// Mitsubishi GX Works2 project: GCP-712CRB_1910022_210518R   PLC: Q03UDV
// SECS

PROGRAM 01INITI
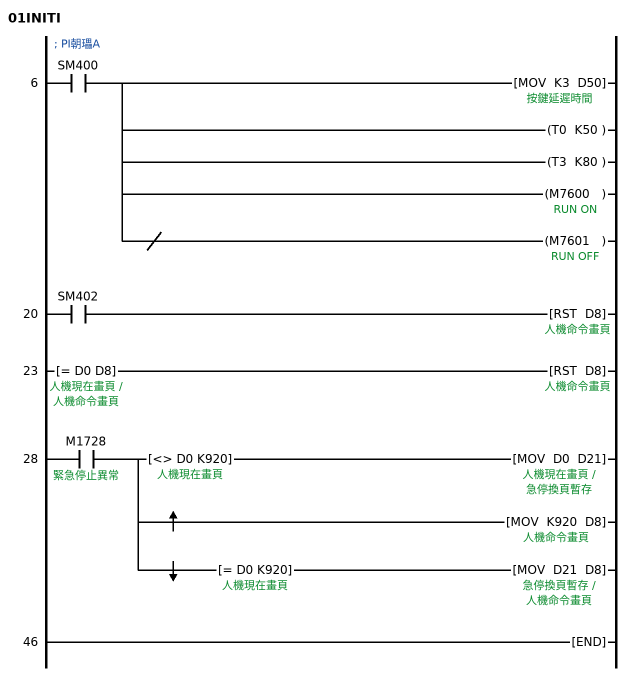
; PI朝瓃Α
6     LD      SM400
      MOV     K3 D50  ; 按鍵延遲時間
      OUT     T0 K50
      OUT     T3 K80
      OUT     M7600  ; RUN ON
      INV
      OUT     M7601  ; RUN OFF
20    LD      SM402
      RST     D8  ; 人機命令畫頁
23    LD=     D0 D8  ; 人機現在畫頁 / 人機命令畫頁
      RST     D8  ; 人機命令畫頁
28    LD      M1728  ; 緊急停止異常
      MPS
      AND<>   D0 K920  ; 人機現在畫頁
      MOV     D0 D21  ; 急停換頁暫存
      MRD
      MEP
      MOV     K920 D8
      MPP
      MEF
      AND=    D0 K920  ; 人機現在畫頁
      MOV     D21 D8
46    END
END_PROGRAM

PROGRAM 02FUNC
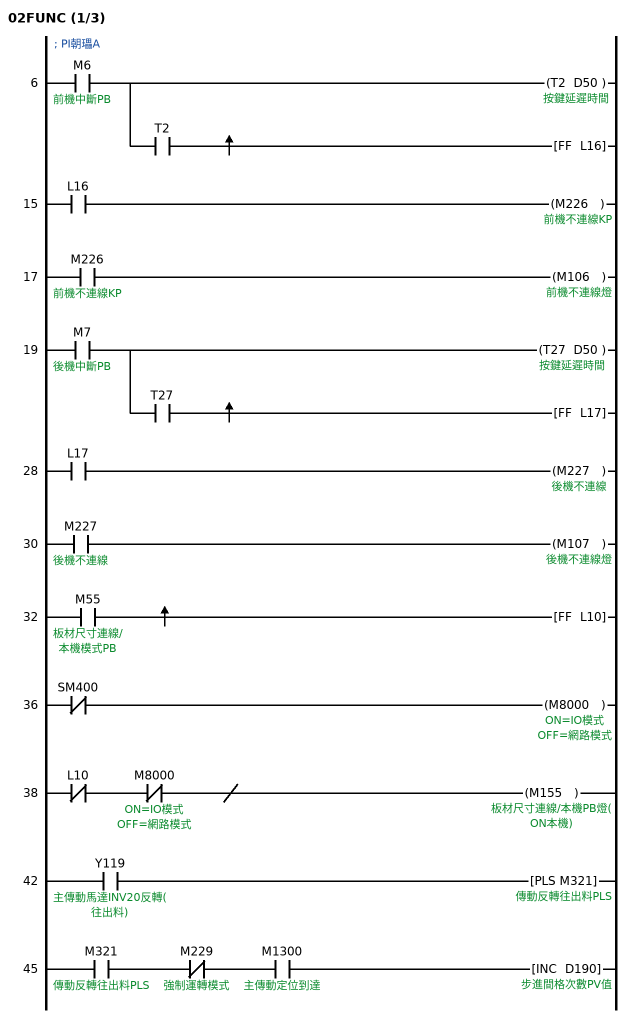
; PI朝瓃Α
6     LD      M6  ; 前機中斷PB
      OUT     T2 D50  ; 按鍵延遲時間
      AND     T2
      MEP
      FF      L16
15    LD      L16
      OUT     M226  ; 前機不連線KP
17    LD      M226  ; 前機不連線KP
      OUT     M106  ; 前機不連線燈
19    LD      M7  ; 後機中斷PB
      OUT     T27 D50  ; 按鍵延遲時間
      AND     T27
      MEP
      FF      L17
28    LD      L17
      OUT     M227  ; 後機不連線
30    LD      M227  ; 後機不連線
      OUT     M107  ; 後機不連線燈
32    LD      M55  ; 板材尺寸連線/本機模式PB
      MEP
      FF      L10
36    LDI     SM400
      OUT     M8000  ; ON=IO模式 OFF=網路模式
38    LDI     L10
      ANI     M8000  ; ON=IO模式 OFF=網路模式
      INV
      OUT     M155  ; 板材尺寸連線/本機PB燈(ON本機)
42    LD      Y119  ; 主傳動馬達INV20反轉(往出料)
      PLS     M321  ; 傳動反轉往出料PLS
45    LD      M321  ; 傳動反轉往出料PLS
      ANI     M229  ; 強制運轉模式
      AND     M1300  ; 主傳動定位到達
      INC     D190  ; 步進間格次數PV值
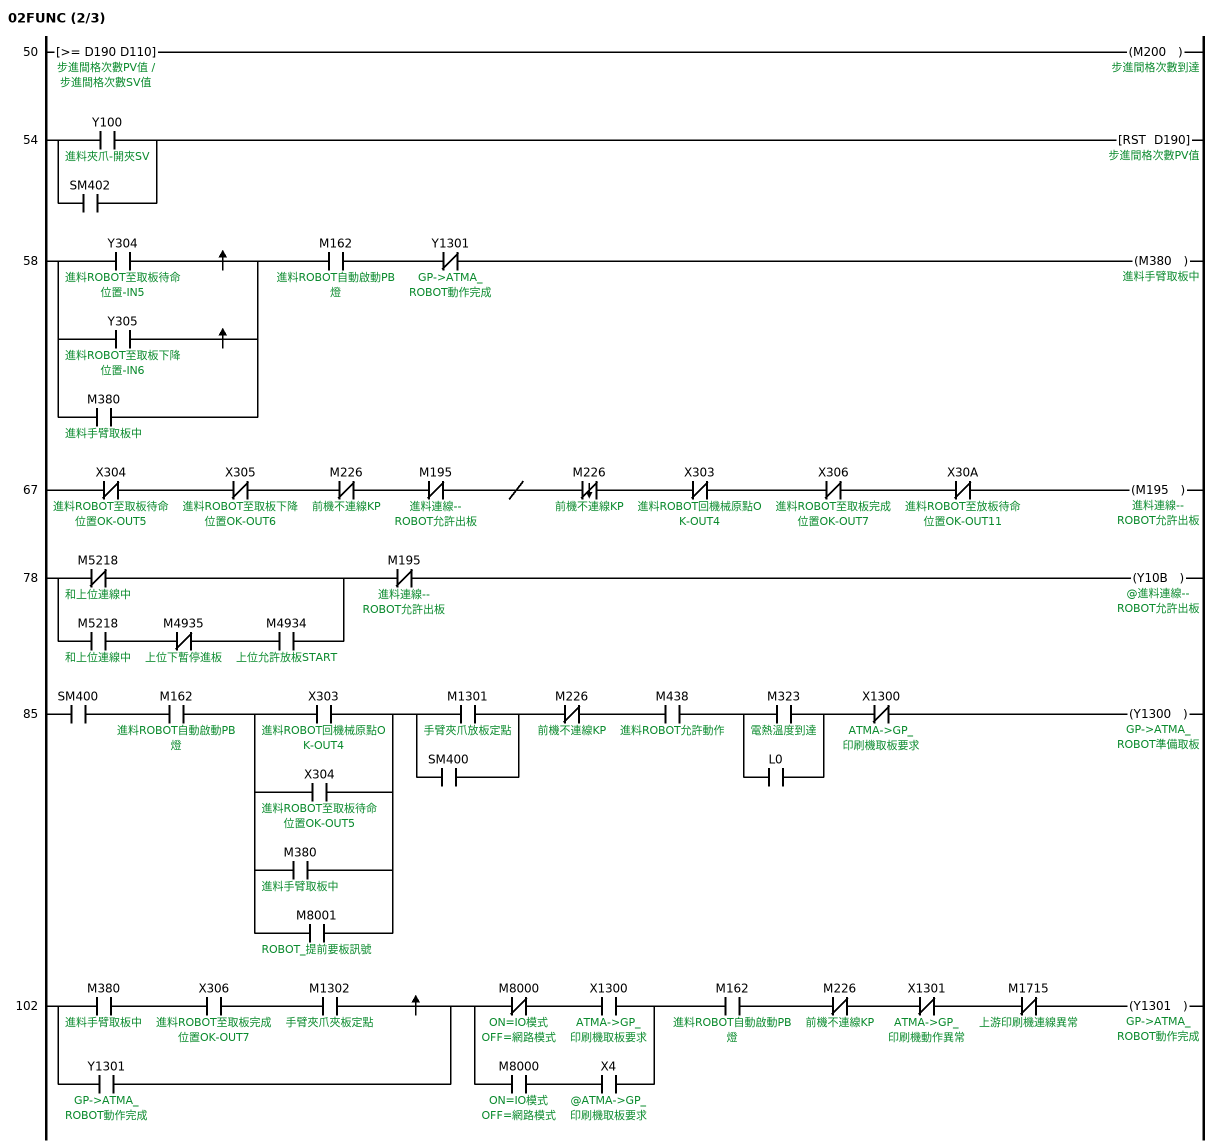
50    LD>=    D190 D110  ; 步進間格次數PV值 / 步進間格次數SV值
      OUT     M200  ; 步進間格次數到達
54    LD      Y100  ; 進料夾爪-開夾SV
      OR      SM402
      RST     D190  ; 步進間格次數PV值
58    LD      Y304  ; 進料ROBOT至取板待命位置-IN5
      MEP
      LD      Y305  ; 進料ROBOT至取板下降位置-IN6
      MEP
      ORB
      OR      M380  ; 進料手臂取板中
      AND     M162  ; 進料ROBOT自動啟動PB燈
      ANI     Y1301  ; GP->ATMA_ROBOT動作完成
      OUT     M380  ; 進料手臂取板中
67    LDI     X304  ; 進料ROBOT至取板待命位置OK-OUT5
      ANI     X305  ; 進料ROBOT至取板下降位置OK-OUT6
      ANI     M226  ; 前機不連線KP
      ANI     M195  ; 進料連線--ROBOT允許出板
      INV
      ANDFI   M226  ; 前機不連線KP
      ANI     X303  ; 進料ROBOT回機械原點OK-OUT4
      ANI     X306  ; 進料ROBOT至取板完成位置OK-OUT7
      ANI     X30A  ; 進料ROBOT至放板待命位置OK-OUT11
      OUT     M195  ; 進料連線--ROBOT允許出板
78    LDI     M5218  ; 和上位連線中
      LD      M5218  ; 和上位連線中
      ANI     M4935  ; 上位下暫停進板
      AND     M4934  ; 上位允許放板START
      ORB
      ANI     M195  ; 進料連線--ROBOT允許出板
      OUT     Y10B  ; @進料連線--ROBOT允許出板
85    LD      SM400
      AND     M162  ; 進料ROBOT自動啟動PB燈
      LD      X303  ; 進料ROBOT回機械原點OK-OUT4
      OR      X304  ; 進料ROBOT至取板待命位置OK-OUT5
      OR      M380  ; 進料手臂取板中
      OR      M8001  ; ROBOT_提前要板訊號
      ANB
      LD      M1301  ; 手臂夾爪放板定點
      OR      SM400
      ANB
      ANI     M226  ; 前機不連線KP
      AND     M438  ; 進料ROBOT允許動作
      LD      M323  ; 電熱溫度到達
      OR      L0
      ANB
      ANI     X1300  ; ATMA->GP_印刷機取板要求
      OUT     Y1300  ; GP->ATMA_ROBOT準備取板
102   LD      M380  ; 進料手臂取板中
      AND     X306  ; 進料ROBOT至取板完成位置OK-OUT7
      AND     M1302  ; 手臂夾爪夾板定點
      MEP
      OR      Y1301  ; GP->ATMA_ROBOT動作完成
      LDI     M8000  ; ON=IO模式 OFF=網路模式
      AND     X1300  ; ATMA->GP_印刷機取板要求
      LD      M8000  ; ON=IO模式 OFF=網路模式
      AND     X4  ; @ATMA->GP_印刷機取板要求
      ORB
      ANB
      AND     M162  ; 進料ROBOT自動啟動PB燈
      ANI     M226  ; 前機不連線KP
      ANI     X1301  ; ATMA->GP_印刷機動作異常
      ANI     M1715  ; 上游印刷機連線異常
      OUT     Y1301  ; GP->ATMA_ROBOT動作完成
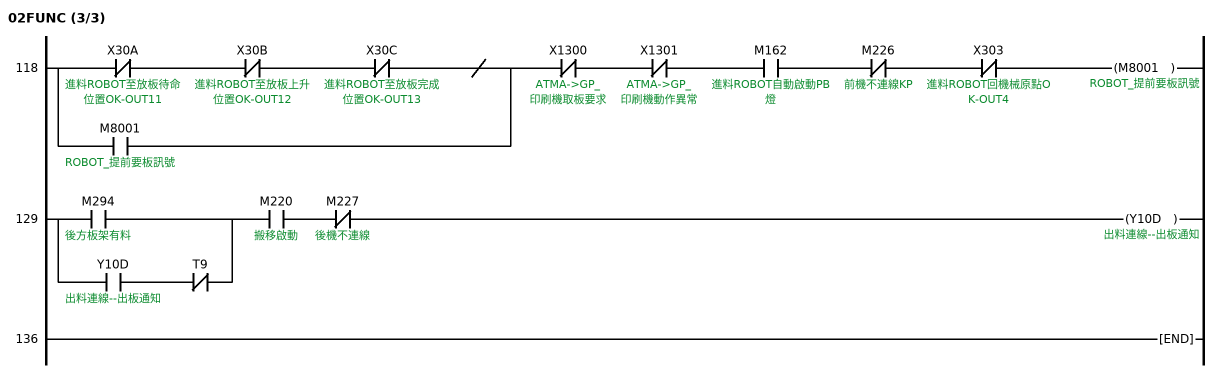
118   LDI     X30A  ; 進料ROBOT至放板待命位置OK-OUT11
      ANI     X30B  ; 進料ROBOT至放板上升位置OK-OUT12
      ANI     X30C  ; 進料ROBOT至放板完成位置OK-OUT13
      INV
      OR      M8001  ; ROBOT_提前要板訊號
      ANI     X1300  ; ATMA->GP_印刷機取板要求
      ANI     X1301  ; ATMA->GP_印刷機動作異常
      AND     M162  ; 進料ROBOT自動啟動PB燈
      ANI     M226  ; 前機不連線KP
      ANI     X303  ; 進料ROBOT回機械原點OK-OUT4
      OUT     M8001  ; ROBOT_提前要板訊號
129   LD      M294  ; 後方板架有料
      LD      Y10D  ; 出料連線--出板通知
      ANI     T9
      ORB
      AND     M220  ; 搬移啟動
      ANI     M227  ; 後機不連線
      OUT     Y10D  ; 出料連線--出板通知
136   END
END_PROGRAM

PROGRAM 03ORIGIN
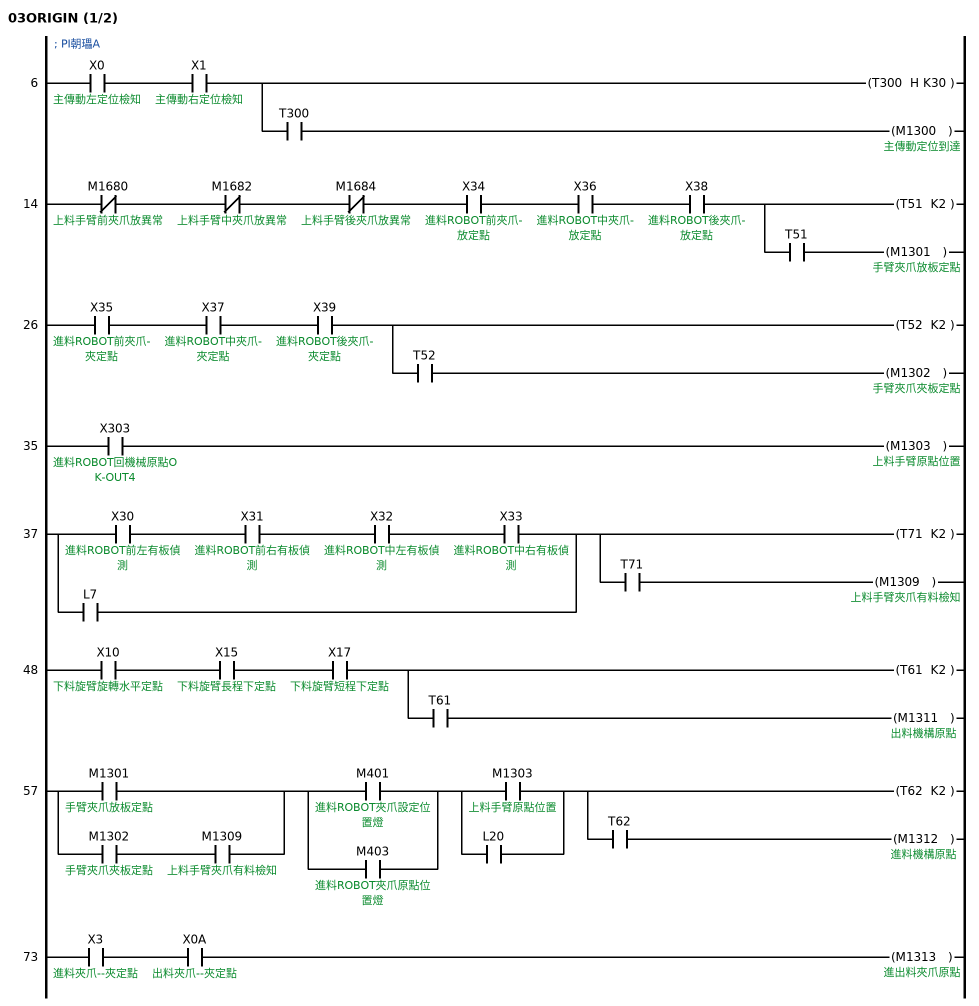
; PI朝瓃Α
6     LD      X0  ; 主傳動左定位檢知
      AND     X1  ; 主傳動右定位檢知
      OUTH    T300 K30
      AND     T300
      OUT     M1300  ; 主傳動定位到達
14    LDI     M1680  ; 上料手臂前夾爪放異常
      ANI     M1682  ; 上料手臂中夾爪放異常
      ANI     M1684  ; 上料手臂後夾爪放異常
      AND     X34  ; 進料ROBOT前夾爪-放定點
      AND     X36  ; 進料ROBOT中夾爪-放定點
      AND     X38  ; 進料ROBOT後夾爪-放定點
      OUT     T51 K2
      AND     T51
      OUT     M1301  ; 手臂夾爪放板定點
26    LD      X35  ; 進料ROBOT前夾爪-夾定點
      AND     X37  ; 進料ROBOT中夾爪-夾定點
      AND     X39  ; 進料ROBOT後夾爪-夾定點
      OUT     T52 K2
      AND     T52
      OUT     M1302  ; 手臂夾爪夾板定點
35    LD      X303  ; 進料ROBOT回機械原點OK-OUT4
      OUT     M1303  ; 上料手臂原點位置
37    LD      X30  ; 進料ROBOT前左有板偵測
      AND     X31  ; 進料ROBOT前右有板偵測
      AND     X32  ; 進料ROBOT中左有板偵測
      AND     X33  ; 進料ROBOT中右有板偵測
      OR      L7
      OUT     T71 K2
      AND     T71
      OUT     M1309  ; 上料手臂夾爪有料檢知
48    LD      X10  ; 下料旋臂旋轉水平定點
      AND     X15  ; 下料旋臂長程下定點
      AND     X17  ; 下料旋臂短程下定點
      OUT     T61 K2
      AND     T61
      OUT     M1311  ; 出料機構原點
57    LD      M1301  ; 手臂夾爪放板定點
      LD      M1302  ; 手臂夾爪夾板定點
      AND     M1309  ; 上料手臂夾爪有料檢知
      ORB
      LD      M401  ; 進料ROBOT夾爪設定位置燈
      OR      M403  ; 進料ROBOT夾爪原點位置燈
      ANB
      LD      M1303  ; 上料手臂原點位置
      OR      L20
      ANB
      OUT     T62 K2
      AND     T62
      OUT     M1312  ; 進料機構原點
73    LD      X3  ; 進料夾爪--夾定點
      AND     X0A  ; 出料夾爪--夾定點
      OUT     M1313  ; 進出料夾爪原點
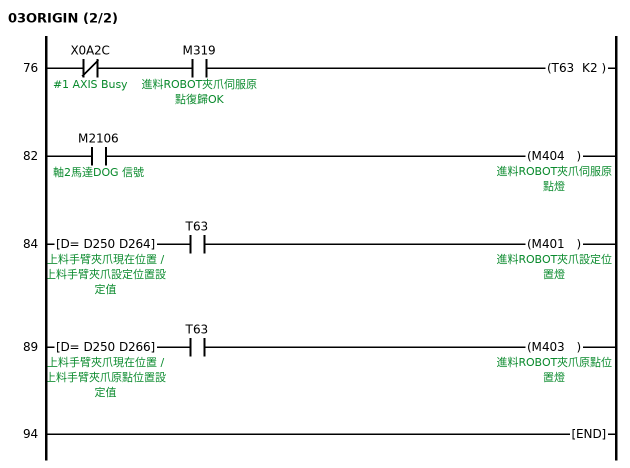
76    LDI     X0A2C  ; #1 AXIS Busy
      AND     M319  ; 進料ROBOT夾爪伺服原點復歸OK
      OUT     T63 K2
82    LD      M2106  ; 軸2馬達DOG 信號
      OUT     M404  ; 進料ROBOT夾爪伺服原點燈
84    LDD=    D250 D264  ; 上料手臂夾爪現在位置 / 上料手臂夾爪設定位置設定值
      AND     T63
      OUT     M401  ; 進料ROBOT夾爪設定位置燈
89    LDD=    D250 D266  ; 上料手臂夾爪現在位置 / 上料手臂夾爪原點位置設定值
      AND     T63
      OUT     M403  ; 進料ROBOT夾爪原點位置燈
94    END
END_PROGRAM

PROGRAM 04LOAD
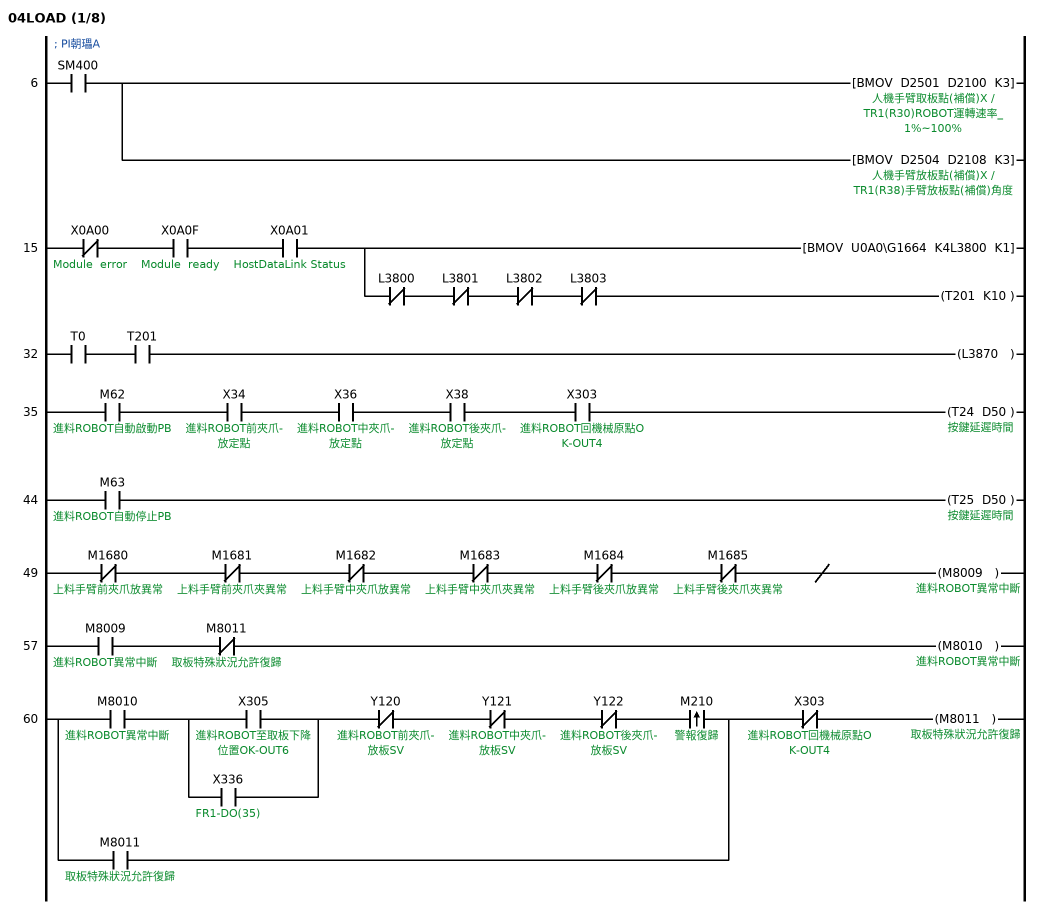
; PI朝瓃Α
6     LD      SM400
      BMOV    D2501 D2100 K3  ; 人機手臂取板點(補償)X / TR1(R30)ROBOT運轉速率_1%~100%
      BMOV    D2504 D2108 K3  ; 人機手臂放板點(補償)X / TR1(R38)手臂放板點(補償)角度
15    LDI     X0A00  ; Module  error
      AND     X0A0F  ; Module  ready
      AND     X0A01  ; HostDataLink Status
      BMOV    U0A0\G1664 K4L3800 K1
      ANI     L3800
      ANI     L3801
      ANI     L3802
      ANI     L3803
      OUT     T201 K10
32    LD      T0
      AND     T201
      OUT     L3870
35    LD      M62  ; 進料ROBOT自動啟動PB
      AND     X34  ; 進料ROBOT前夾爪-放定點
      AND     X36  ; 進料ROBOT中夾爪-放定點
      AND     X38  ; 進料ROBOT後夾爪-放定點
      AND     X303  ; 進料ROBOT回機械原點OK-OUT4
      OUT     T24 D50  ; 按鍵延遲時間
44    LD      M63  ; 進料ROBOT自動停止PB
      OUT     T25 D50  ; 按鍵延遲時間
49    LDI     M1680  ; 上料手臂前夾爪放異常
      ANI     M1681  ; 上料手臂前夾爪夾異常
      ANI     M1682  ; 上料手臂中夾爪放異常
      ANI     M1683  ; 上料手臂中夾爪夾異常
      ANI     M1684  ; 上料手臂後夾爪放異常
      ANI     M1685  ; 上料手臂後夾爪夾異常
      INV
      OUT     M8009  ; 進料ROBOT異常中斷
57    LD      M8009  ; 進料ROBOT異常中斷
      ANI     M8011  ; 取板特殊狀況允許復歸
      OUT     M8010  ; 進料ROBOT異常中斷
60    LD      M8010  ; 進料ROBOT異常中斷
      LD      X305  ; 進料ROBOT至取板下降位置OK-OUT6
      OR      X336  ; FR1-DO(35)
      ANB
      ANI     Y120  ; 進料ROBOT前夾爪-放板SV
      ANI     Y121  ; 進料ROBOT中夾爪-放板SV
      ANI     Y122  ; 進料ROBOT後夾爪-放板SV
      ANDP    M210  ; 警報復歸
      OR      M8011  ; 取板特殊狀況允許復歸
      ANI     X303  ; 進料ROBOT回機械原點OK-OUT4
      OUT     M8011  ; 取板特殊狀況允許復歸
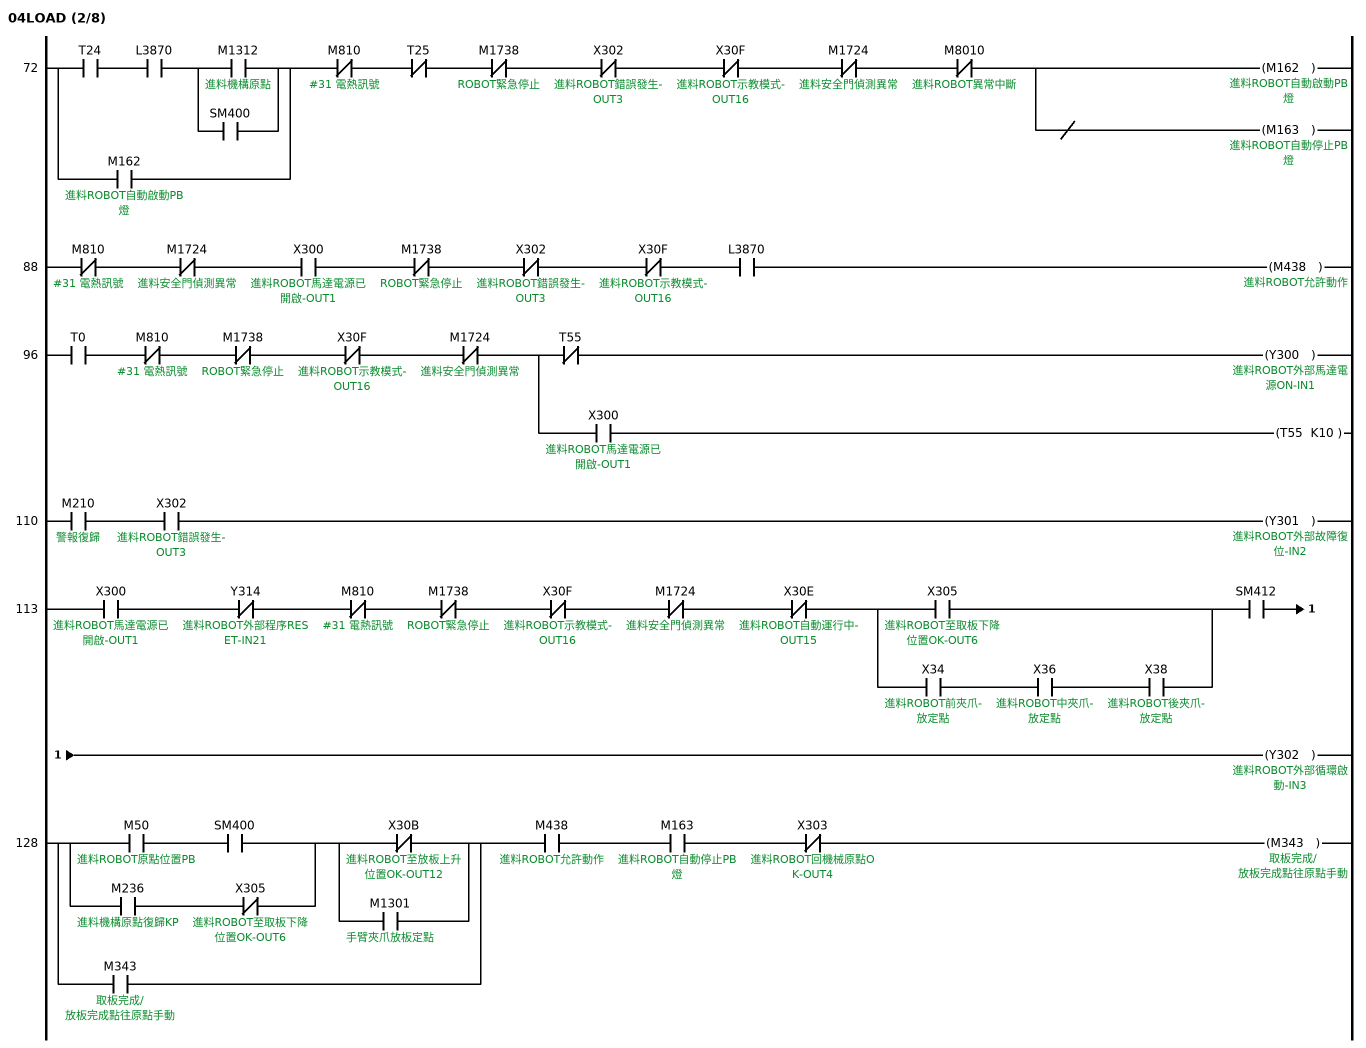
72    LD      T24
      AND     L3870
      LD      M1312  ; 進料機構原點
      OR      SM400
      ANB
      OR      M162  ; 進料ROBOT自動啟動PB燈
      ANI     M810  ; #31 電熱訊號
      ANI     T25
      ANI     M1738  ; ROBOT緊急停止
      ANI     X302  ; 進料ROBOT錯誤發生-OUT3
      ANI     X30F  ; 進料ROBOT示教模式-OUT16
      ANI     M1724  ; 進料安全門偵測異常
      ANI     M8010  ; 進料ROBOT異常中斷
      OUT     M162  ; 進料ROBOT自動啟動PB燈
      INV
      OUT     M163  ; 進料ROBOT自動停止PB燈
88    LDI     M810  ; #31 電熱訊號
      ANI     M1724  ; 進料安全門偵測異常
      AND     X300  ; 進料ROBOT馬達電源已開啟-OUT1
      ANI     M1738  ; ROBOT緊急停止
      ANI     X302  ; 進料ROBOT錯誤發生-OUT3
      ANI     X30F  ; 進料ROBOT示教模式-OUT16
      AND     L3870
      OUT     M438  ; 進料ROBOT允許動作
96    LD      T0
      ANI     M810  ; #31 電熱訊號
      ANI     M1738  ; ROBOT緊急停止
      ANI     X30F  ; 進料ROBOT示教模式-OUT16
      ANI     M1724  ; 進料安全門偵測異常
      MPS
      ANI     T55
      OUT     Y300  ; 進料ROBOT外部馬達電源ON-IN1
      MPP
      AND     X300  ; 進料ROBOT馬達電源已開啟-OUT1
      OUT     T55 K10
110   LD      M210  ; 警報復歸
      AND     X302  ; 進料ROBOT錯誤發生-OUT3
      OUT     Y301  ; 進料ROBOT外部故障復位-IN2
113   LD      X300  ; 進料ROBOT馬達電源已開啟-OUT1
      ANI     Y314  ; 進料ROBOT外部程序RESET-IN21
      ANI     M810  ; #31 電熱訊號
      ANI     M1738  ; ROBOT緊急停止
      ANI     X30F  ; 進料ROBOT示教模式-OUT16
      ANI     M1724  ; 進料安全門偵測異常
      ANI     X30E  ; 進料ROBOT自動運行中-OUT15
      LD      X305  ; 進料ROBOT至取板下降位置OK-OUT6
      LD      X34  ; 進料ROBOT前夾爪-放定點
      AND     X36  ; 進料ROBOT中夾爪-放定點
      AND     X38  ; 進料ROBOT後夾爪-放定點
      ORB
      ANB
      AND     SM412
      OUT     Y302  ; 進料ROBOT外部循環啟動-IN3
128   LD      M50  ; 進料ROBOT原點位置PB
      AND     SM400
      LD      M236  ; 進料機構原點復歸KP
      ANI     X305  ; 進料ROBOT至取板下降位置OK-OUT6
      ORB
      LDI     X30B  ; 進料ROBOT至放板上升位置OK-OUT12
      OR      M1301  ; 手臂夾爪放板定點
      ANB
      OR      M343  ; 取板完成/放板完成點往原點手動
      AND     M438  ; 進料ROBOT允許動作
      AND     M163  ; 進料ROBOT自動停止PB燈
      ANI     X303  ; 進料ROBOT回機械原點OK-OUT4
      OUT     M343  ; 取板完成/放板完成點往原點手動
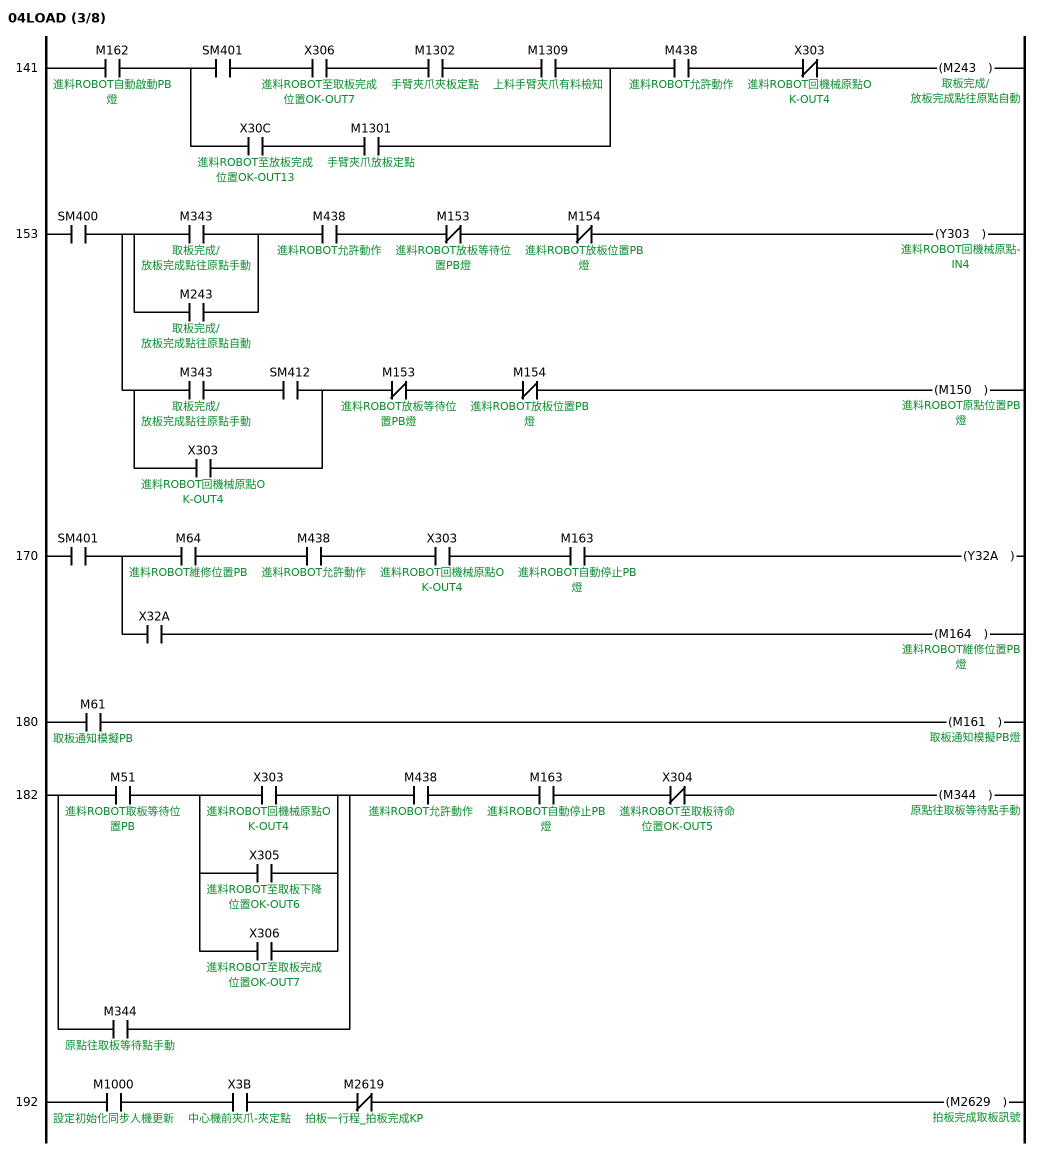
141   LD      M162  ; 進料ROBOT自動啟動PB燈
      LD      SM401
      AND     X306  ; 進料ROBOT至取板完成位置OK-OUT7
      AND     M1302  ; 手臂夾爪夾板定點
      AND     M1309  ; 上料手臂夾爪有料檢知
      LD      X30C  ; 進料ROBOT至放板完成位置OK-OUT13
      AND     M1301  ; 手臂夾爪放板定點
      ORB
      ANB
      AND     M438  ; 進料ROBOT允許動作
      ANI     X303  ; 進料ROBOT回機械原點OK-OUT4
      OUT     M243  ; 取板完成/放板完成點往原點自動
153   LD      SM400
      MPS
      LD      M343  ; 取板完成/放板完成點往原點手動
      OR      M243  ; 取板完成/放板完成點往原點自動
      ANB
      AND     M438  ; 進料ROBOT允許動作
      ANI     M153  ; 進料ROBOT放板等待位置PB燈
      ANI     M154  ; 進料ROBOT放板位置PB燈
      OUT     Y303  ; 進料ROBOT回機械原點-IN4
      MPP
      LD      M343  ; 取板完成/放板完成點往原點手動
      AND     SM412
      OR      X303  ; 進料ROBOT回機械原點OK-OUT4
      ANB
      ANI     M153  ; 進料ROBOT放板等待位置PB燈
      ANI     M154  ; 進料ROBOT放板位置PB燈
      OUT     M150  ; 進料ROBOT原點位置PB燈
170   LD      SM401
      MPS
      AND     M64  ; 進料ROBOT維修位置PB
      AND     M438  ; 進料ROBOT允許動作
      AND     X303  ; 進料ROBOT回機械原點OK-OUT4
      AND     M163  ; 進料ROBOT自動停止PB燈
      OUT     Y32A
      MPP
      AND     X32A
      OUT     M164  ; 進料ROBOT維修位置PB燈
180   LD      M61  ; 取板通知模擬PB
      OUT     M161  ; 取板通知模擬PB燈
182   LD      M51  ; 進料ROBOT取板等待位置PB
      LD      X303  ; 進料ROBOT回機械原點OK-OUT4
      OR      X305  ; 進料ROBOT至取板下降位置OK-OUT6
      OR      X306  ; 進料ROBOT至取板完成位置OK-OUT7
      ANB
      OR      M344  ; 原點往取板等待點手動
      AND     M438  ; 進料ROBOT允許動作
      AND     M163  ; 進料ROBOT自動停止PB燈
      ANI     X304  ; 進料ROBOT至取板待命位置OK-OUT5
      OUT     M344  ; 原點往取板等待點手動
192   LD      M1000  ; 設定初始化同步人機更新
      AND     X3B  ; 中心機前夾爪-夾定點
      ANI     M2619  ; 拍板一行程_拍板完成KP
      OUT     M2629  ; 拍板完成取板訊號
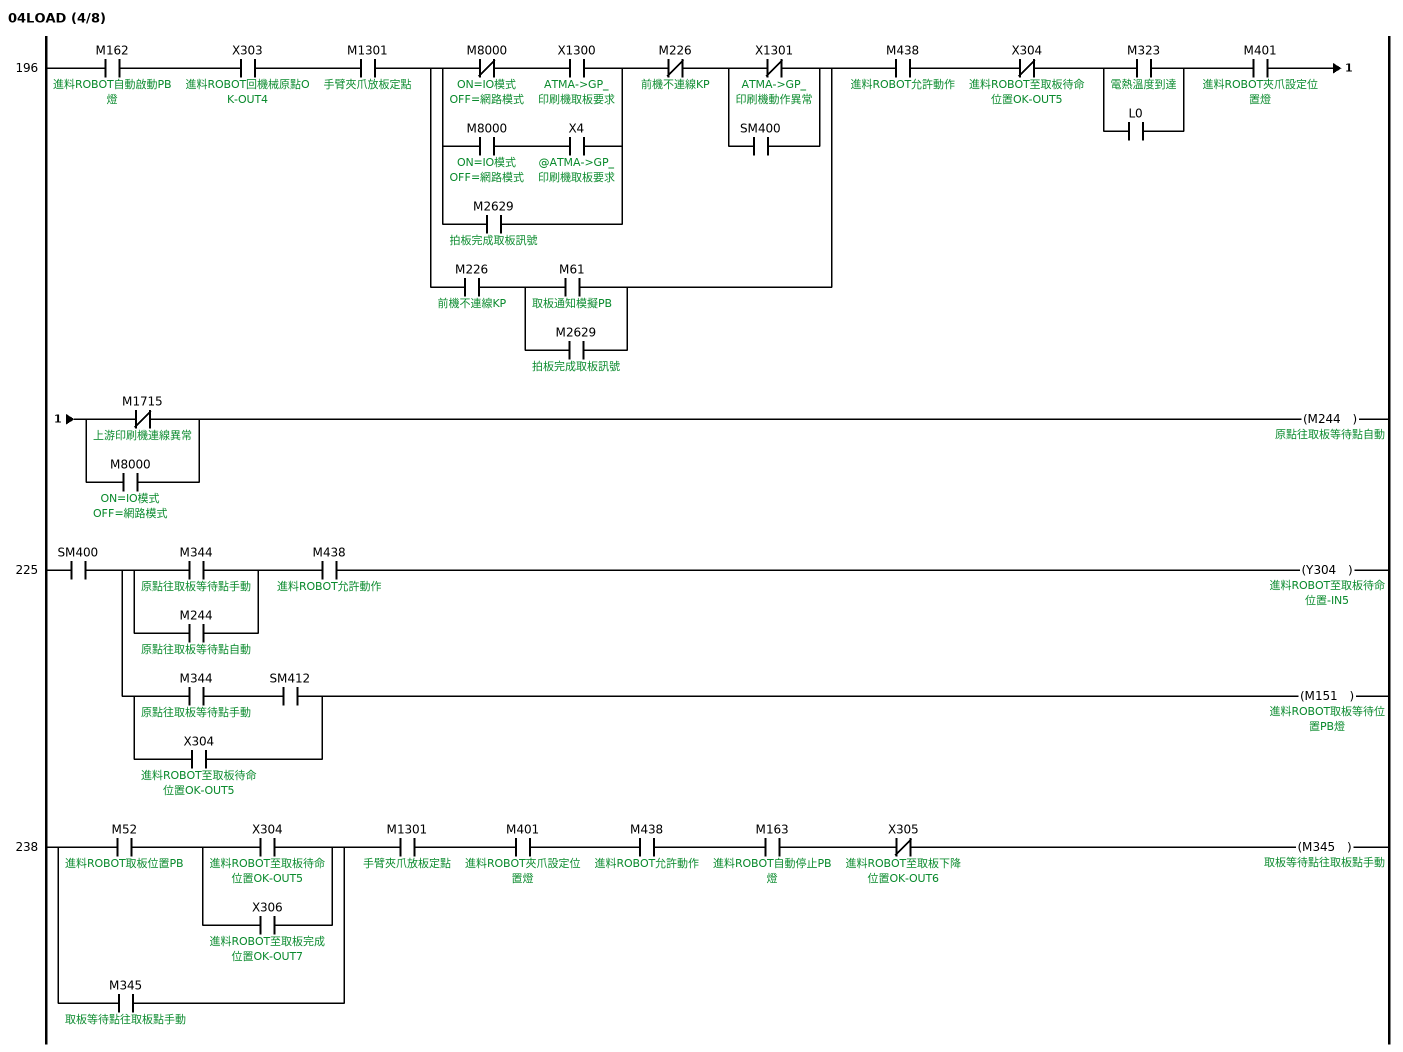
196   LD      M162  ; 進料ROBOT自動啟動PB燈
      AND     X303  ; 進料ROBOT回機械原點OK-OUT4
      AND     M1301  ; 手臂夾爪放板定點
      LDI     M8000  ; ON=IO模式 OFF=網路模式
      AND     X1300  ; ATMA->GP_印刷機取板要求
      LD      M8000  ; ON=IO模式 OFF=網路模式
      AND     X4  ; @ATMA->GP_印刷機取板要求
      ORB
      OR      M2629  ; 拍板完成取板訊號
      ANI     M226  ; 前機不連線KP
      LDI     X1301  ; ATMA->GP_印刷機動作異常
      OR      SM400
      ANB
      LD      M226  ; 前機不連線KP
      LD      M61  ; 取板通知模擬PB
      OR      M2629  ; 拍板完成取板訊號
      ANB
      ORB
      ANB
      AND     M438  ; 進料ROBOT允許動作
      ANI     X304  ; 進料ROBOT至取板待命位置OK-OUT5
      LD      M323  ; 電熱溫度到達
      OR      L0
      ANB
      AND     M401  ; 進料ROBOT夾爪設定位置燈
      LDI     M1715  ; 上游印刷機連線異常
      OR      M8000  ; ON=IO模式 OFF=網路模式
      ANB
      OUT     M244  ; 原點往取板等待點自動
225   LD      SM400
      MPS
      LD      M344  ; 原點往取板等待點手動
      OR      M244  ; 原點往取板等待點自動
      ANB
      AND     M438  ; 進料ROBOT允許動作
      OUT     Y304  ; 進料ROBOT至取板待命位置-IN5
      MPP
      LD      M344  ; 原點往取板等待點手動
      AND     SM412
      OR      X304  ; 進料ROBOT至取板待命位置OK-OUT5
      ANB
      OUT     M151  ; 進料ROBOT取板等待位置PB燈
238   LD      M52  ; 進料ROBOT取板位置PB
      LD      X304  ; 進料ROBOT至取板待命位置OK-OUT5
      OR      X306  ; 進料ROBOT至取板完成位置OK-OUT7
      ANB
      OR      M345  ; 取板等待點往取板點手動
      AND     M1301  ; 手臂夾爪放板定點
      AND     M401  ; 進料ROBOT夾爪設定位置燈
      AND     M438  ; 進料ROBOT允許動作
      AND     M163  ; 進料ROBOT自動停止PB燈
      ANI     X305  ; 進料ROBOT至取板下降位置OK-OUT6
      OUT     M345  ; 取板等待點往取板點手動
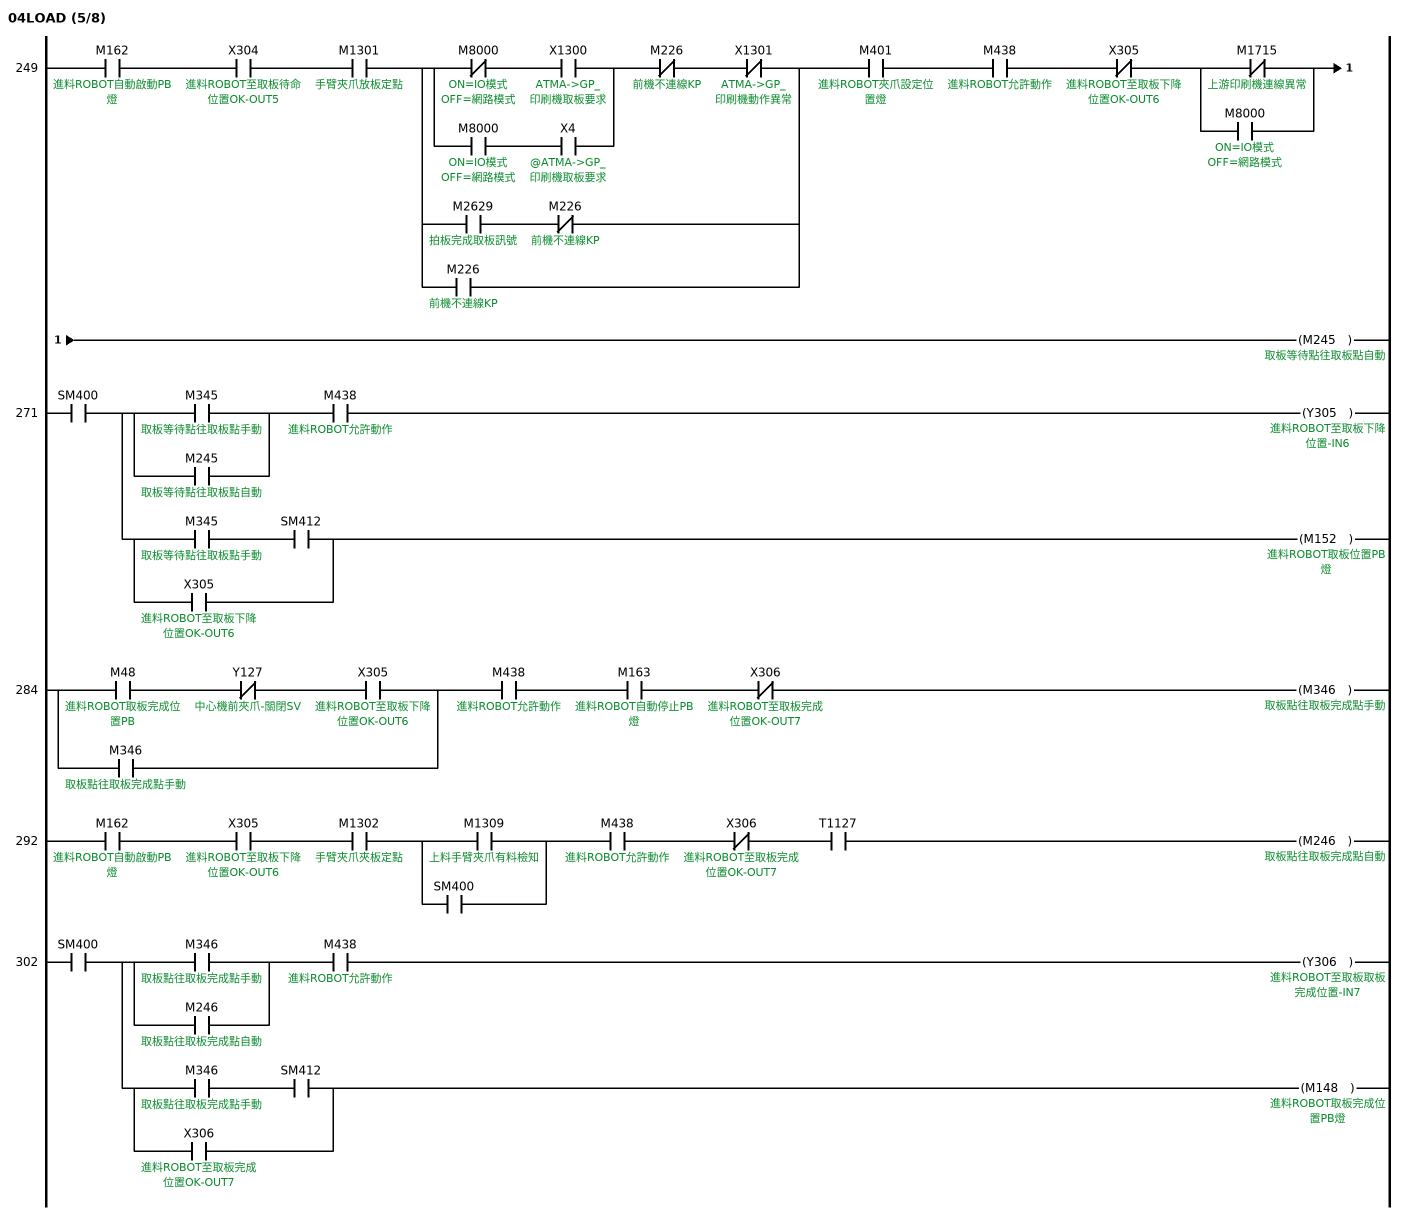
249   LD      M162  ; 進料ROBOT自動啟動PB燈
      AND     X304  ; 進料ROBOT至取板待命位置OK-OUT5
      AND     M1301  ; 手臂夾爪放板定點
      LDI     M8000  ; ON=IO模式 OFF=網路模式
      AND     X1300  ; ATMA->GP_印刷機取板要求
      LD      M8000  ; ON=IO模式 OFF=網路模式
      AND     X4  ; @ATMA->GP_印刷機取板要求
      ORB
      ANI     M226  ; 前機不連線KP
      ANI     X1301  ; ATMA->GP_印刷機動作異常
      LD      M2629  ; 拍板完成取板訊號
      ANI     M226  ; 前機不連線KP
      ORB
      OR      M226  ; 前機不連線KP
      ANB
      AND     M401  ; 進料ROBOT夾爪設定位置燈
      AND     M438  ; 進料ROBOT允許動作
      ANI     X305  ; 進料ROBOT至取板下降位置OK-OUT6
      LDI     M1715  ; 上游印刷機連線異常
      OR      M8000  ; ON=IO模式 OFF=網路模式
      ANB
      OUT     M245  ; 取板等待點往取板點自動
271   LD      SM400
      MPS
      LD      M345  ; 取板等待點往取板點手動
      OR      M245  ; 取板等待點往取板點自動
      ANB
      AND     M438  ; 進料ROBOT允許動作
      OUT     Y305  ; 進料ROBOT至取板下降位置-IN6
      MPP
      LD      M345  ; 取板等待點往取板點手動
      AND     SM412
      OR      X305  ; 進料ROBOT至取板下降位置OK-OUT6
      ANB
      OUT     M152  ; 進料ROBOT取板位置PB燈
284   LD      M48  ; 進料ROBOT取板完成位置PB
      ANI     Y127  ; 中心機前夾爪-關閉SV
      AND     X305  ; 進料ROBOT至取板下降位置OK-OUT6
      OR      M346  ; 取板點往取板完成點手動
      AND     M438  ; 進料ROBOT允許動作
      AND     M163  ; 進料ROBOT自動停止PB燈
      ANI     X306  ; 進料ROBOT至取板完成位置OK-OUT7
      OUT     M346  ; 取板點往取板完成點手動
292   LD      M162  ; 進料ROBOT自動啟動PB燈
      AND     X305  ; 進料ROBOT至取板下降位置OK-OUT6
      AND     M1302  ; 手臂夾爪夾板定點
      LD      M1309  ; 上料手臂夾爪有料檢知
      OR      SM400
      ANB
      AND     M438  ; 進料ROBOT允許動作
      ANI     X306  ; 進料ROBOT至取板完成位置OK-OUT7
      AND     T1127
      OUT     M246  ; 取板點往取板完成點自動
302   LD      SM400
      MPS
      LD      M346  ; 取板點往取板完成點手動
      OR      M246  ; 取板點往取板完成點自動
      ANB
      AND     M438  ; 進料ROBOT允許動作
      OUT     Y306  ; 進料ROBOT至取板取板完成位置-IN7
      MPP
      LD      M346  ; 取板點往取板完成點手動
      AND     SM412
      OR      X306  ; 進料ROBOT至取板完成位置OK-OUT7
      ANB
      OUT     M148  ; 進料ROBOT取板完成位置PB燈
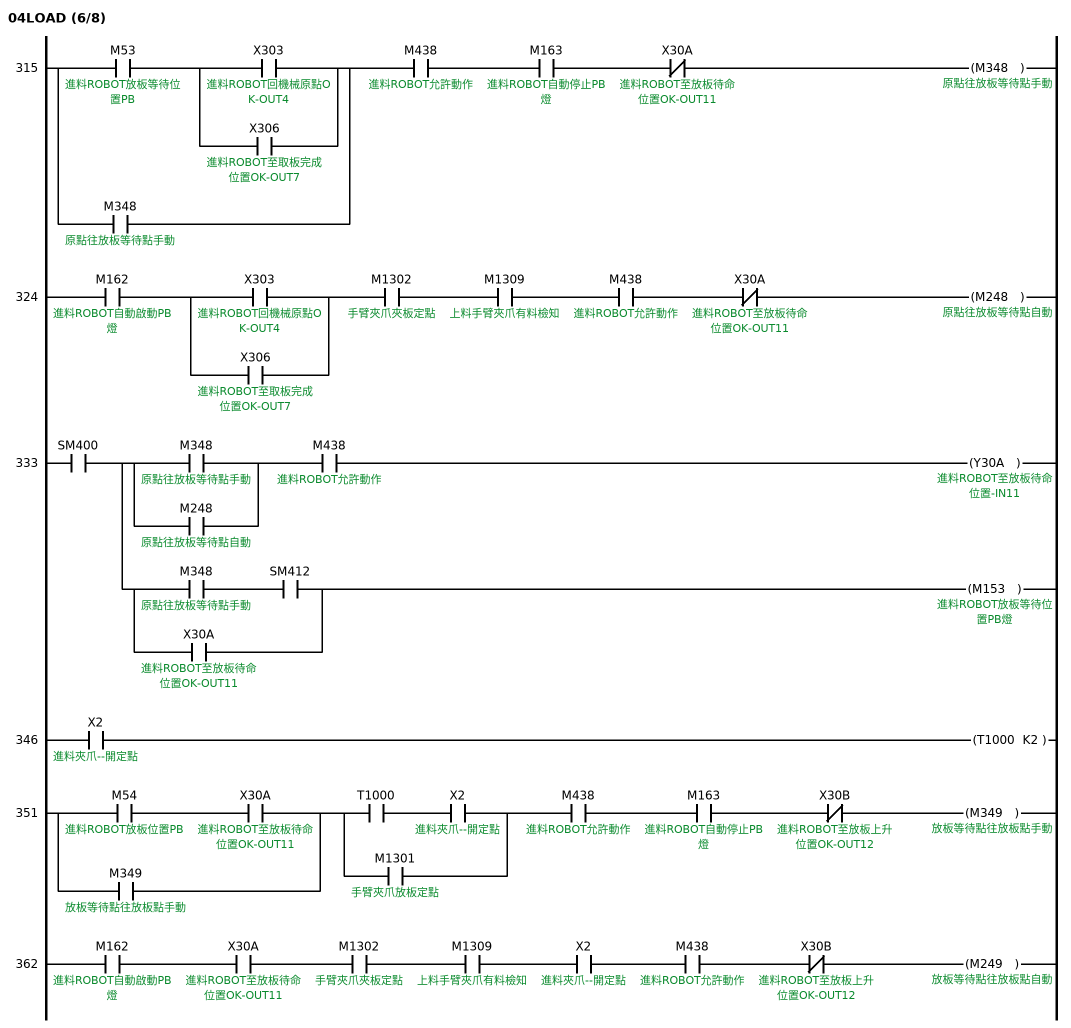
315   LD      M53  ; 進料ROBOT放板等待位置PB
      LD      X303  ; 進料ROBOT回機械原點OK-OUT4
      OR      X306  ; 進料ROBOT至取板完成位置OK-OUT7
      ANB
      OR      M348  ; 原點往放板等待點手動
      AND     M438  ; 進料ROBOT允許動作
      AND     M163  ; 進料ROBOT自動停止PB燈
      ANI     X30A  ; 進料ROBOT至放板待命位置OK-OUT11
      OUT     M348  ; 原點往放板等待點手動
324   LD      M162  ; 進料ROBOT自動啟動PB燈
      LD      X303  ; 進料ROBOT回機械原點OK-OUT4
      OR      X306  ; 進料ROBOT至取板完成位置OK-OUT7
      ANB
      AND     M1302  ; 手臂夾爪夾板定點
      AND     M1309  ; 上料手臂夾爪有料檢知
      AND     M438  ; 進料ROBOT允許動作
      ANI     X30A  ; 進料ROBOT至放板待命位置OK-OUT11
      OUT     M248  ; 原點往放板等待點自動
333   LD      SM400
      MPS
      LD      M348  ; 原點往放板等待點手動
      OR      M248  ; 原點往放板等待點自動
      ANB
      AND     M438  ; 進料ROBOT允許動作
      OUT     Y30A  ; 進料ROBOT至放板待命位置-IN11
      MPP
      LD      M348  ; 原點往放板等待點手動
      AND     SM412
      OR      X30A  ; 進料ROBOT至放板待命位置OK-OUT11
      ANB
      OUT     M153  ; 進料ROBOT放板等待位置PB燈
346   LD      X2  ; 進料夾爪--開定點
      OUT     T1000 K2
351   LD      M54  ; 進料ROBOT放板位置PB
      AND     X30A  ; 進料ROBOT至放板待命位置OK-OUT11
      OR      M349  ; 放板等待點往放板點手動
      LD      T1000
      AND     X2  ; 進料夾爪--開定點
      OR      M1301  ; 手臂夾爪放板定點
      ANB
      AND     M438  ; 進料ROBOT允許動作
      AND     M163  ; 進料ROBOT自動停止PB燈
      ANI     X30B  ; 進料ROBOT至放板上升位置OK-OUT12
      OUT     M349  ; 放板等待點往放板點手動
362   LD      M162  ; 進料ROBOT自動啟動PB燈
      AND     X30A  ; 進料ROBOT至放板待命位置OK-OUT11
      AND     M1302  ; 手臂夾爪夾板定點
      AND     M1309  ; 上料手臂夾爪有料檢知
      AND     X2  ; 進料夾爪--開定點
      AND     M438  ; 進料ROBOT允許動作
      ANI     X30B  ; 進料ROBOT至放板上升位置OK-OUT12
      OUT     M249  ; 放板等待點往放板點自動
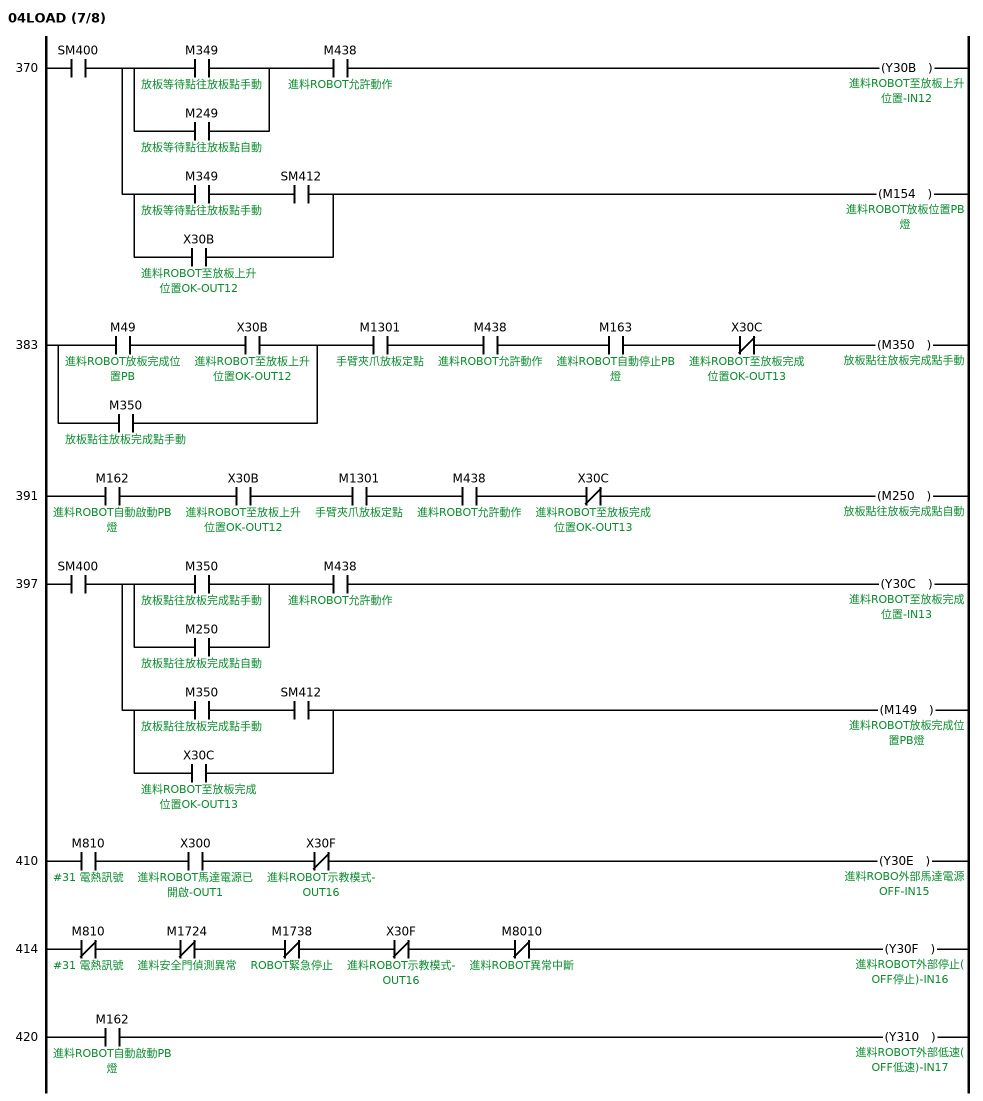
370   LD      SM400
      MPS
      LD      M349  ; 放板等待點往放板點手動
      OR      M249  ; 放板等待點往放板點自動
      ANB
      AND     M438  ; 進料ROBOT允許動作
      OUT     Y30B  ; 進料ROBOT至放板上升位置-IN12
      MPP
      LD      M349  ; 放板等待點往放板點手動
      AND     SM412
      OR      X30B  ; 進料ROBOT至放板上升位置OK-OUT12
      ANB
      OUT     M154  ; 進料ROBOT放板位置PB燈
383   LD      M49  ; 進料ROBOT放板完成位置PB
      AND     X30B  ; 進料ROBOT至放板上升位置OK-OUT12
      OR      M350  ; 放板點往放板完成點手動
      AND     M1301  ; 手臂夾爪放板定點
      AND     M438  ; 進料ROBOT允許動作
      AND     M163  ; 進料ROBOT自動停止PB燈
      ANI     X30C  ; 進料ROBOT至放板完成位置OK-OUT13
      OUT     M350  ; 放板點往放板完成點手動
391   LD      M162  ; 進料ROBOT自動啟動PB燈
      AND     X30B  ; 進料ROBOT至放板上升位置OK-OUT12
      AND     M1301  ; 手臂夾爪放板定點
      AND     M438  ; 進料ROBOT允許動作
      ANI     X30C  ; 進料ROBOT至放板完成位置OK-OUT13
      OUT     M250  ; 放板點往放板完成點自動
397   LD      SM400
      MPS
      LD      M350  ; 放板點往放板完成點手動
      OR      M250  ; 放板點往放板完成點自動
      ANB
      AND     M438  ; 進料ROBOT允許動作
      OUT     Y30C  ; 進料ROBOT至放板完成位置-IN13
      MPP
      LD      M350  ; 放板點往放板完成點手動
      AND     SM412
      OR      X30C  ; 進料ROBOT至放板完成位置OK-OUT13
      ANB
      OUT     M149  ; 進料ROBOT放板完成位置PB燈
410   LD      M810  ; #31 電熱訊號
      AND     X300  ; 進料ROBOT馬達電源已開啟-OUT1
      ANI     X30F  ; 進料ROBOT示教模式-OUT16
      OUT     Y30E  ; 進料ROBO外部馬達電源OFF-IN15
414   LDI     M810  ; #31 電熱訊號
      ANI     M1724  ; 進料安全門偵測異常
      ANI     M1738  ; ROBOT緊急停止
      ANI     X30F  ; 進料ROBOT示教模式-OUT16
      ANI     M8010  ; 進料ROBOT異常中斷
      OUT     Y30F  ; 進料ROBOT外部停止(OFF停止)-IN16
420   LD      M162  ; 進料ROBOT自動啟動PB燈
      OUT     Y310  ; 進料ROBOT外部低速(OFF低速)-IN17
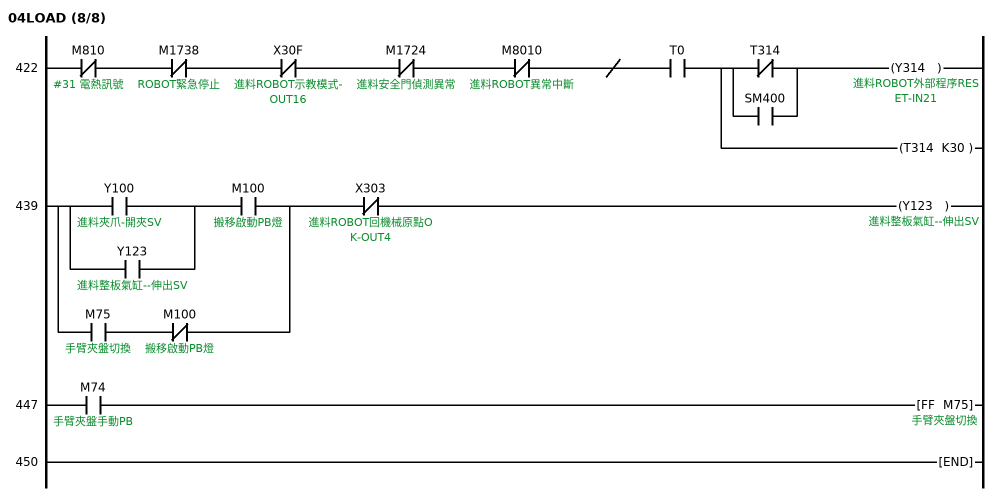
422   LDI     M810  ; #31 電熱訊號
      ANI     M1738  ; ROBOT緊急停止
      ANI     X30F  ; 進料ROBOT示教模式-OUT16
      ANI     M1724  ; 進料安全門偵測異常
      ANI     M8010  ; 進料ROBOT異常中斷
      INV
      AND     T0
      MPS
      LDI     T314
      OR      SM400
      ANB
      OUT     Y314  ; 進料ROBOT外部程序RESET-IN21
      MPP
      OUT     T314 K30
439   LD      Y100  ; 進料夾爪-開夾SV
      OR      Y123  ; 進料整板氣缸--伸出SV
      AND     M100  ; 搬移啟動PB燈
      LD      M75  ; 手臂夾盤切換
      ANI     M100  ; 搬移啟動PB燈
      ORB
      ANI     X303  ; 進料ROBOT回機械原點OK-OUT4
      OUT     Y123  ; 進料整板氣缸--伸出SV
447   LD      M74  ; 手臂夾盤手動PB
      FF      M75
450   END
END_PROGRAM

PROGRAM 05LOADUP
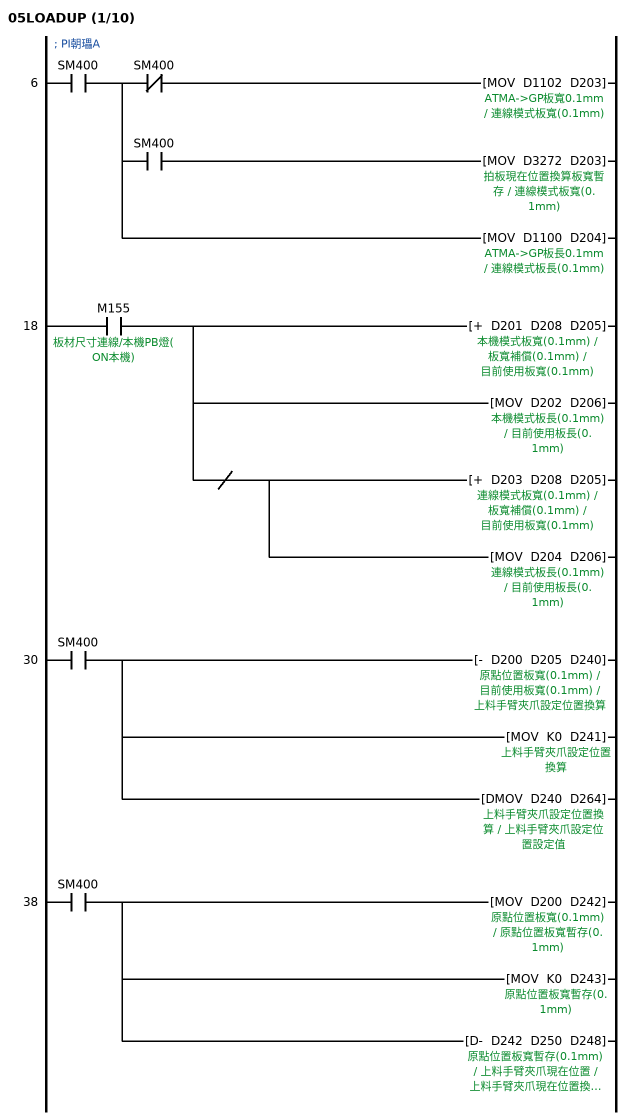
; PI朝瓃Α
6     LD      SM400
      MPS
      ANI     SM400
      MOV     D1102 D203  ; ATMA->GP板寬0.1mm / 連線模式板寬(0.1mm)
      MRD
      AND     SM400
      MOV     D3272 D203  ; 拍板現在位置換算板寬暫存
      MPP
      MOV     D1100 D204  ; ATMA->GP板長0.1mm / 連線模式板長(0.1mm)
18    LD      M155  ; 板材尺寸連線/本機PB燈(ON本機)
      +       D201 D208 D205  ; 本機模式板寬(0.1mm) / 板寬補償(0.1mm) / 目前使用板寬(0.1mm)
      MOV     D202 D206  ; 本機模式板長(0.1mm) / 目前使用板長(0.1mm)
      INV
      +       D203 D208 D205
      MOV     D204 D206
30    LD      SM400
      -       D200 D205 D240  ; 原點位置板寬(0.1mm) / 上料手臂夾爪設定位置換算
      MOV     K0 D241  ; 上料手臂夾爪設定位置換算
      DMOV    D240 D264  ; 上料手臂夾爪設定位置設定值
38    LD      SM400
      MOV     D200 D242  ; 原點位置板寬暫存(0.1mm)
      MOV     K0 D243  ; 原點位置板寬暫存(0.1mm)
      D-      D242 D250 D248  ; 上料手臂夾爪現在位置 / 上料手臂夾爪現在位置換算板寬
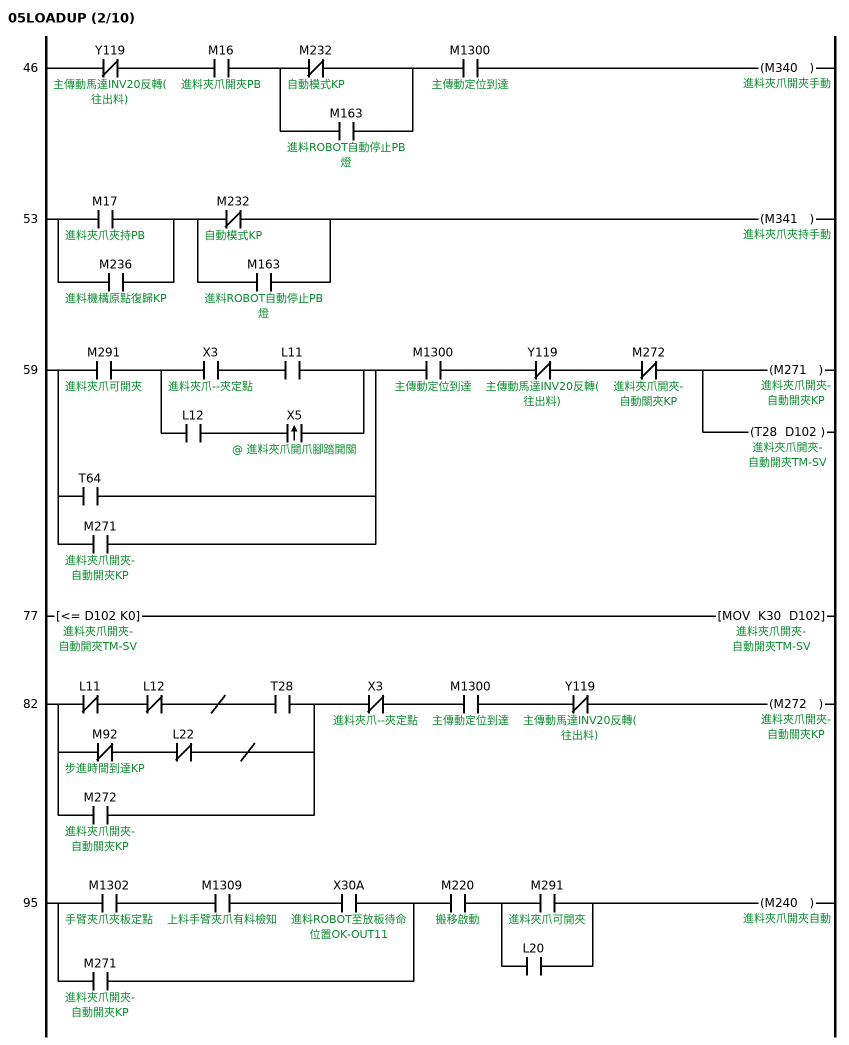
46    LDI     Y119  ; 主傳動馬達INV20反轉(往出料)
      AND     M16  ; 進料夾爪開夾PB
      LDI     M232  ; 自動模式KP
      OR      M163  ; 進料ROBOT自動停止PB燈
      ANB
      AND     M1300  ; 主傳動定位到達
      OUT     M340  ; 進料夾爪開夾手動
53    LD      M17  ; 進料夾爪夾持PB
      OR      M236  ; 進料機構原點復歸KP
      LDI     M232  ; 自動模式KP
      OR      M163  ; 進料ROBOT自動停止PB燈
      ANB
      OUT     M341  ; 進料夾爪夾持手動
59    LD      M291  ; 進料夾爪可開夾
      LD      X3  ; 進料夾爪--夾定點
      AND     L11
      LD      L12
      ANDP    X5  ; @ 進料夾爪開爪腳踏開關
      ORB
      ANB
      OR      T64
      OR      M271  ; 進料夾爪開夾-自動開夾KP
      AND     M1300  ; 主傳動定位到達
      ANI     Y119  ; 主傳動馬達INV20反轉(往出料)
      ANI     M272  ; 進料夾爪開夾-自動關夾KP
      OUT     M271  ; 進料夾爪開夾-自動開夾KP
      OUT     T28 D102  ; 進料夾爪開夾-自動開夾TM-SV
77    LD<=    D102 K0  ; 進料夾爪開夾-自動開夾TM-SV
      MOV     K30 D102
82    LDI     L11
      ANI     L12
      INV
      AND     T28
      LDI     M92  ; 步進時間到達KP
      ANI     L22
      INV
      ORB
      OR      M272  ; 進料夾爪開夾-自動關夾KP
      ANI     X3  ; 進料夾爪--夾定點
      AND     M1300  ; 主傳動定位到達
      ANI     Y119  ; 主傳動馬達INV20反轉(往出料)
      OUT     M272  ; 進料夾爪開夾-自動關夾KP
95    LD      M1302  ; 手臂夾爪夾板定點
      AND     M1309  ; 上料手臂夾爪有料檢知
      AND     X30A  ; 進料ROBOT至放板待命位置OK-OUT11
      OR      M271  ; 進料夾爪開夾-自動開夾KP
      AND     M220  ; 搬移啟動
      LD      M291  ; 進料夾爪可開夾
      OR      L20
      ANB
      OUT     M240  ; 進料夾爪開夾自動
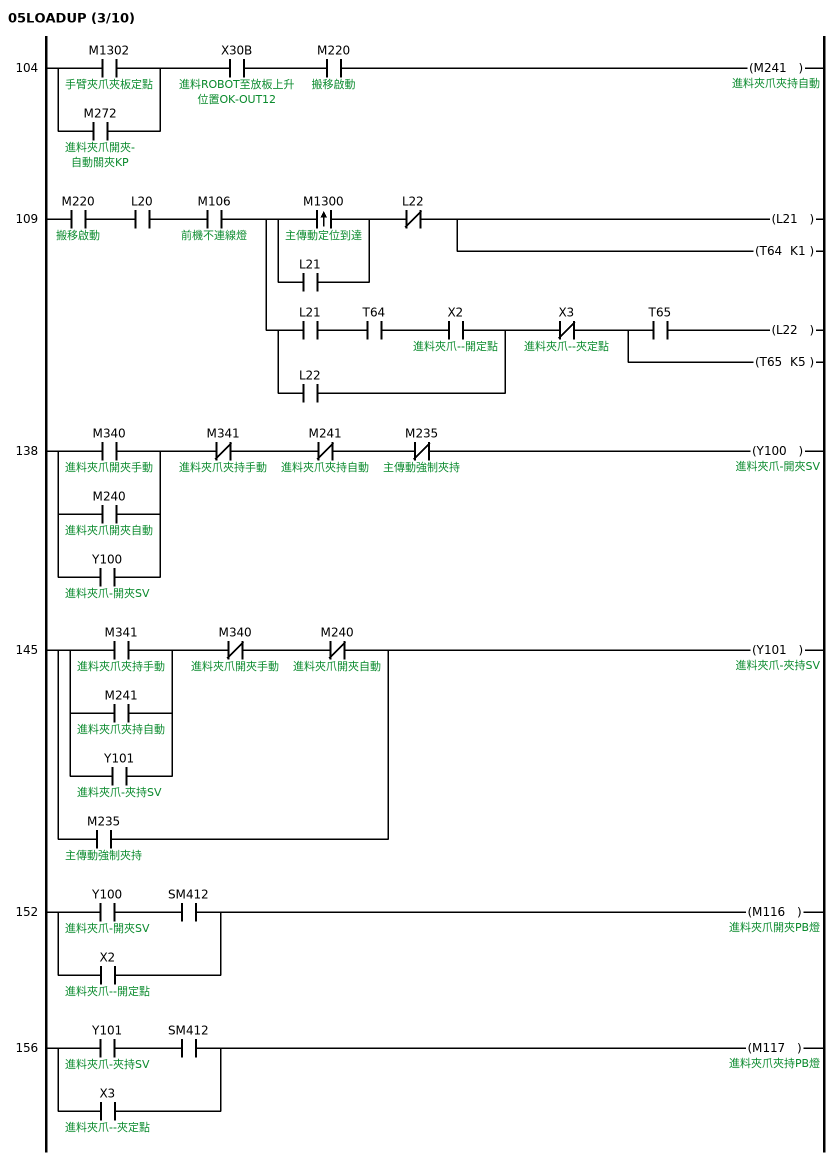
104   LD      M1302  ; 手臂夾爪夾板定點
      OR      M272  ; 進料夾爪開夾-自動關夾KP
      AND     X30B  ; 進料ROBOT至放板上升位置OK-OUT12
      AND     M220  ; 搬移啟動
      OUT     M241  ; 進料夾爪夾持自動
109   LD      M220  ; 搬移啟動
      AND     L20
      AND     M106  ; 前機不連線燈
      MPS
      LDP     M1300  ; 主傳動定位到達
      OR      L21
      ANB
      ANI     L22
      OUT     L21
      OUT     T64 K1
      MPP
      LD      L21
      AND     T64
      AND     X2  ; 進料夾爪--開定點
      OR      L22
      ANB
      ANI     X3  ; 進料夾爪--夾定點
      MPS
      AND     T65
      OUT     L22
      MPP
      OUT     T65 K5
138   LD      M340  ; 進料夾爪開夾手動
      OR      M240  ; 進料夾爪開夾自動
      OR      Y100  ; 進料夾爪-開夾SV
      ANI     M341  ; 進料夾爪夾持手動
      ANI     M241  ; 進料夾爪夾持自動
      ANI     M235  ; 主傳動強制夾持
      OUT     Y100  ; 進料夾爪-開夾SV
145   LD      M341  ; 進料夾爪夾持手動
      OR      M241  ; 進料夾爪夾持自動
      OR      Y101  ; 進料夾爪-夾持SV
      ANI     M340  ; 進料夾爪開夾手動
      ANI     M240  ; 進料夾爪開夾自動
      OR      M235  ; 主傳動強制夾持
      OUT     Y101  ; 進料夾爪-夾持SV
152   LD      Y100  ; 進料夾爪-開夾SV
      AND     SM412
      OR      X2  ; 進料夾爪--開定點
      OUT     M116  ; 進料夾爪開夾PB燈
156   LD      Y101  ; 進料夾爪-夾持SV
      AND     SM412
      OR      X3  ; 進料夾爪--夾定點
      OUT     M117  ; 進料夾爪夾持PB燈
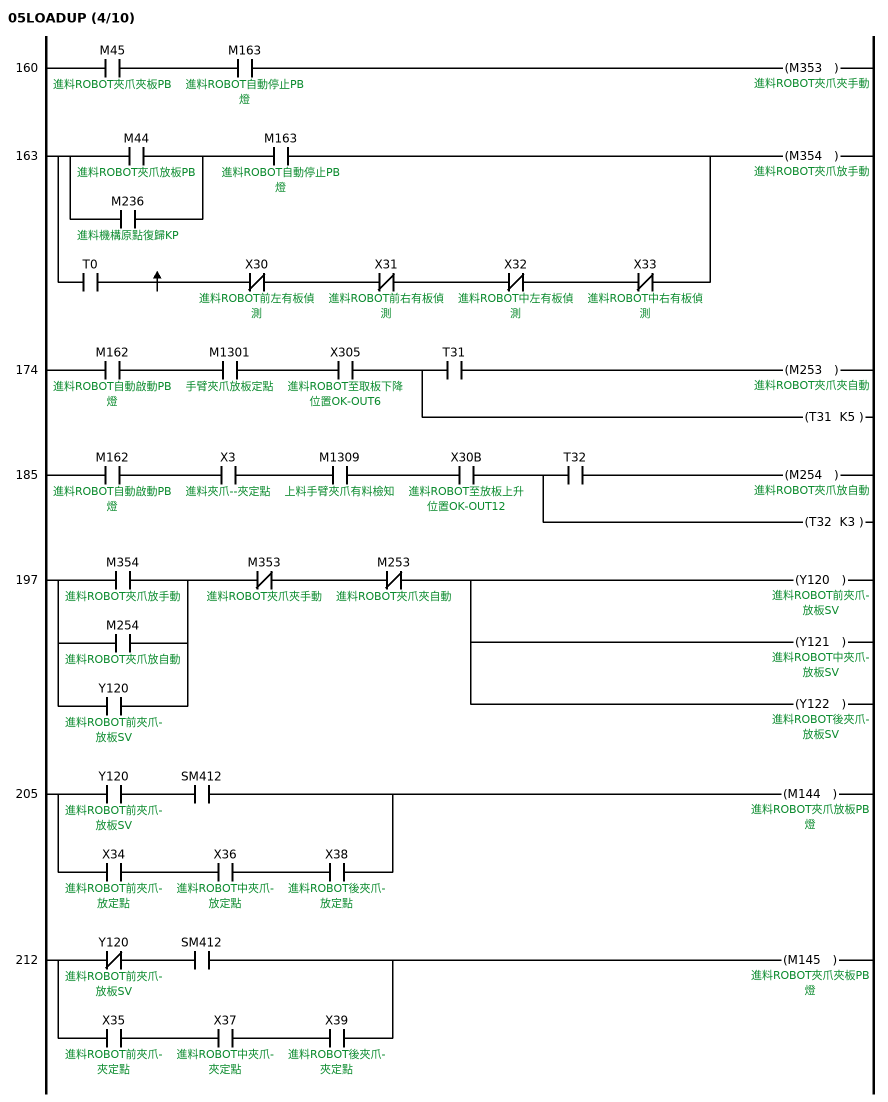
160   LD      M45  ; 進料ROBOT夾爪夾板PB
      AND     M163  ; 進料ROBOT自動停止PB燈
      OUT     M353  ; 進料ROBOT夾爪夾手動
163   LD      M44  ; 進料ROBOT夾爪放板PB
      OR      M236  ; 進料機構原點復歸KP
      AND     M163  ; 進料ROBOT自動停止PB燈
      LD      T0
      MEP
      ANI     X30  ; 進料ROBOT前左有板偵測
      ANI     X31  ; 進料ROBOT前右有板偵測
      ANI     X32  ; 進料ROBOT中左有板偵測
      ANI     X33  ; 進料ROBOT中右有板偵測
      ORB
      OUT     M354  ; 進料ROBOT夾爪放手動
174   LD      M162  ; 進料ROBOT自動啟動PB燈
      AND     M1301  ; 手臂夾爪放板定點
      AND     X305  ; 進料ROBOT至取板下降位置OK-OUT6
      MPS
      AND     T31
      OUT     M253  ; 進料ROBOT夾爪夾自動
      MPP
      OUT     T31 K5
185   LD      M162  ; 進料ROBOT自動啟動PB燈
      AND     X3  ; 進料夾爪--夾定點
      AND     M1309  ; 上料手臂夾爪有料檢知
      AND     X30B  ; 進料ROBOT至放板上升位置OK-OUT12
      MPS
      AND     T32
      OUT     M254  ; 進料ROBOT夾爪放自動
      MPP
      OUT     T32 K3
197   LD      M354  ; 進料ROBOT夾爪放手動
      OR      M254  ; 進料ROBOT夾爪放自動
      OR      Y120  ; 進料ROBOT前夾爪-放板SV
      ANI     M353  ; 進料ROBOT夾爪夾手動
      ANI     M253  ; 進料ROBOT夾爪夾自動
      OUT     Y120  ; 進料ROBOT前夾爪-放板SV
      OUT     Y121  ; 進料ROBOT中夾爪-放板SV
      OUT     Y122  ; 進料ROBOT後夾爪-放板SV
205   LD      Y120  ; 進料ROBOT前夾爪-放板SV
      AND     SM412
      LD      X34  ; 進料ROBOT前夾爪-放定點
      AND     X36  ; 進料ROBOT中夾爪-放定點
      AND     X38  ; 進料ROBOT後夾爪-放定點
      ORB
      OUT     M144  ; 進料ROBOT夾爪放板PB燈
212   LDI     Y120  ; 進料ROBOT前夾爪-放板SV
      AND     SM412
      LD      X35  ; 進料ROBOT前夾爪-夾定點
      AND     X37  ; 進料ROBOT中夾爪-夾定點
      AND     X39  ; 進料ROBOT後夾爪-夾定點
      ORB
      OUT     M145  ; 進料ROBOT夾爪夾板PB燈
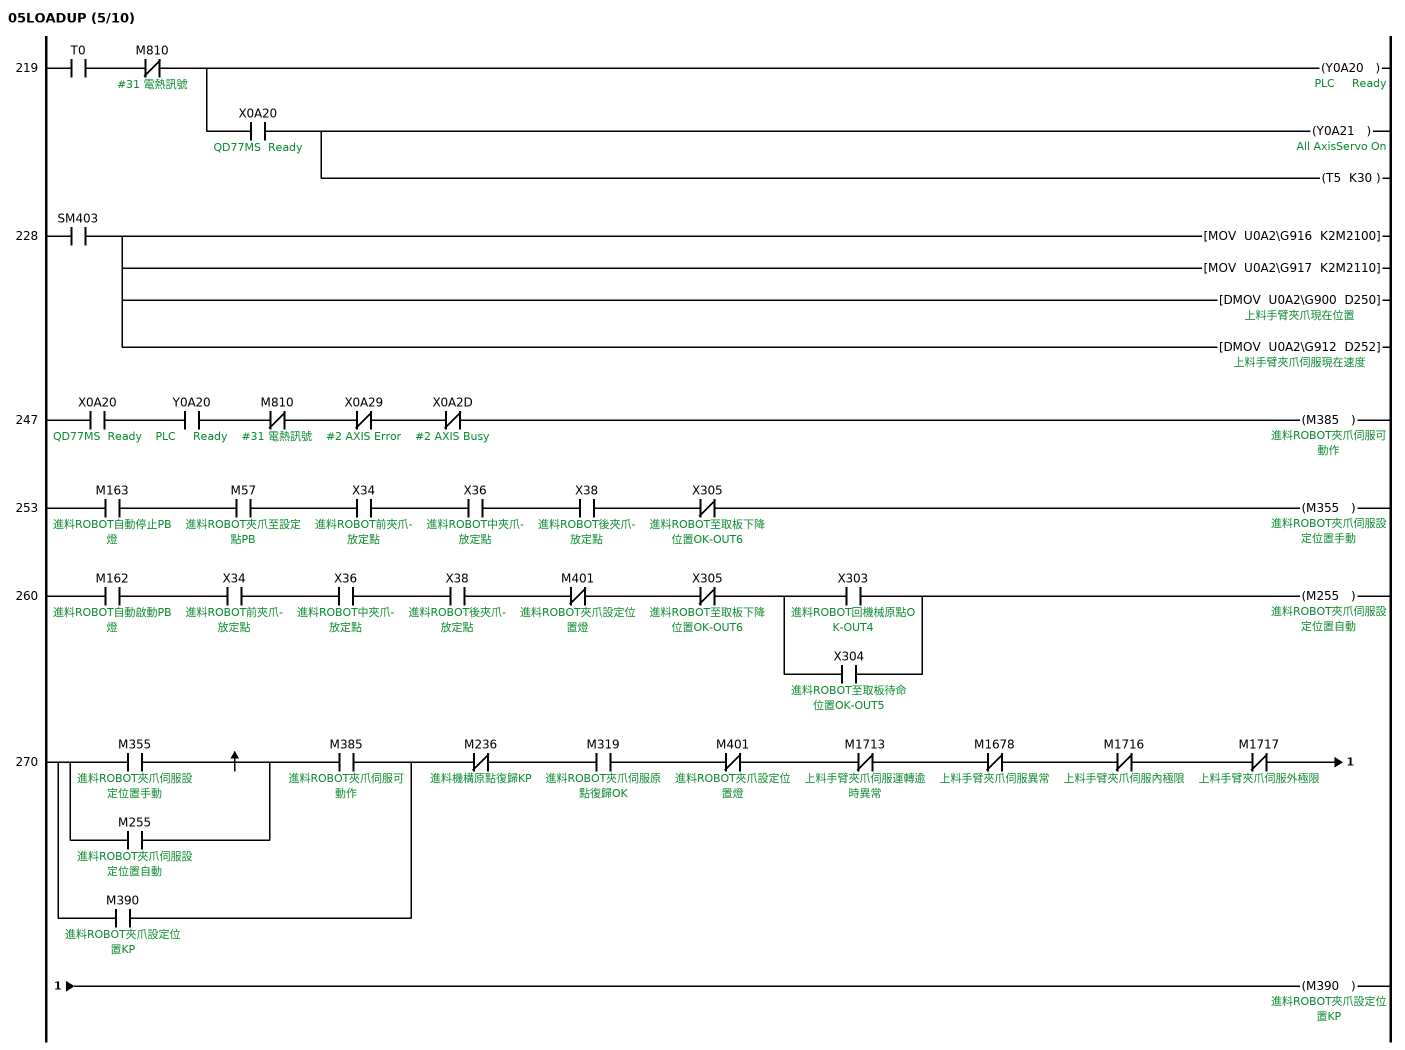
219   LD      T0
      ANI     M810  ; #31 電熱訊號
      OUT     Y0A20  ; PLC     Ready
      AND     X0A20  ; QD77MS  Ready
      OUT     Y0A21  ; All AxisServo On
      OUT     T5 K30
228   LD      SM403
      MOV     U0A2\G916 K2M2100  ; 軸2伺服馬達外極限
      MOV     U0A2\G917 K2M2110  ; Axis02  速度控制
      DMOV    U0A2\G900 D250
      DMOV    U0A2\G912 D252  ; 上料手臂夾爪伺服現在速度
247   LD      X0A20  ; QD77MS  Ready
      AND     Y0A20  ; PLC     Ready
      ANI     M810  ; #31 電熱訊號
      ANI     X0A29  ; #2 AXIS Error
      ANI     X0A2D  ; #2 AXIS Busy
      OUT     M385  ; 進料ROBOT夾爪伺服可動作
253   LD      M163  ; 進料ROBOT自動停止PB燈
      AND     M57  ; 進料ROBOT夾爪至設定點PB
      AND     X34  ; 進料ROBOT前夾爪-放定點
      AND     X36  ; 進料ROBOT中夾爪-放定點
      AND     X38  ; 進料ROBOT後夾爪-放定點
      ANI     X305  ; 進料ROBOT至取板下降位置OK-OUT6
      OUT     M355  ; 進料ROBOT夾爪伺服設定位置手動
260   LD      M162  ; 進料ROBOT自動啟動PB燈
      AND     X34  ; 進料ROBOT前夾爪-放定點
      AND     X36  ; 進料ROBOT中夾爪-放定點
      AND     X38  ; 進料ROBOT後夾爪-放定點
      ANI     M401  ; 進料ROBOT夾爪設定位置燈
      ANI     X305  ; 進料ROBOT至取板下降位置OK-OUT6
      LD      X303  ; 進料ROBOT回機械原點OK-OUT4
      OR      X304  ; 進料ROBOT至取板待命位置OK-OUT5
      ANB
      OUT     M255  ; 進料ROBOT夾爪伺服設定位置自動
270   LD      M355  ; 進料ROBOT夾爪伺服設定位置手動
      MEP
      OR      M255  ; 進料ROBOT夾爪伺服設定位置自動
      AND     M385  ; 進料ROBOT夾爪伺服可動作
      OR      M390  ; 進料ROBOT夾爪設定位置KP
      ANI     M236  ; 進料機構原點復歸KP
      AND     M319  ; 進料ROBOT夾爪伺服原點復歸OK
      ANI     M401  ; 進料ROBOT夾爪設定位置燈
      ANI     M1713  ; 上料手臂夾爪伺服運轉逾時異常
      ANI     M1678  ; 上料手臂夾爪伺服異常
      ANI     M1716  ; 上料手臂夾爪伺服內極限
      ANI     M1717  ; 上料手臂夾爪伺服外極限
      OUT     M390  ; 進料ROBOT夾爪設定位置KP
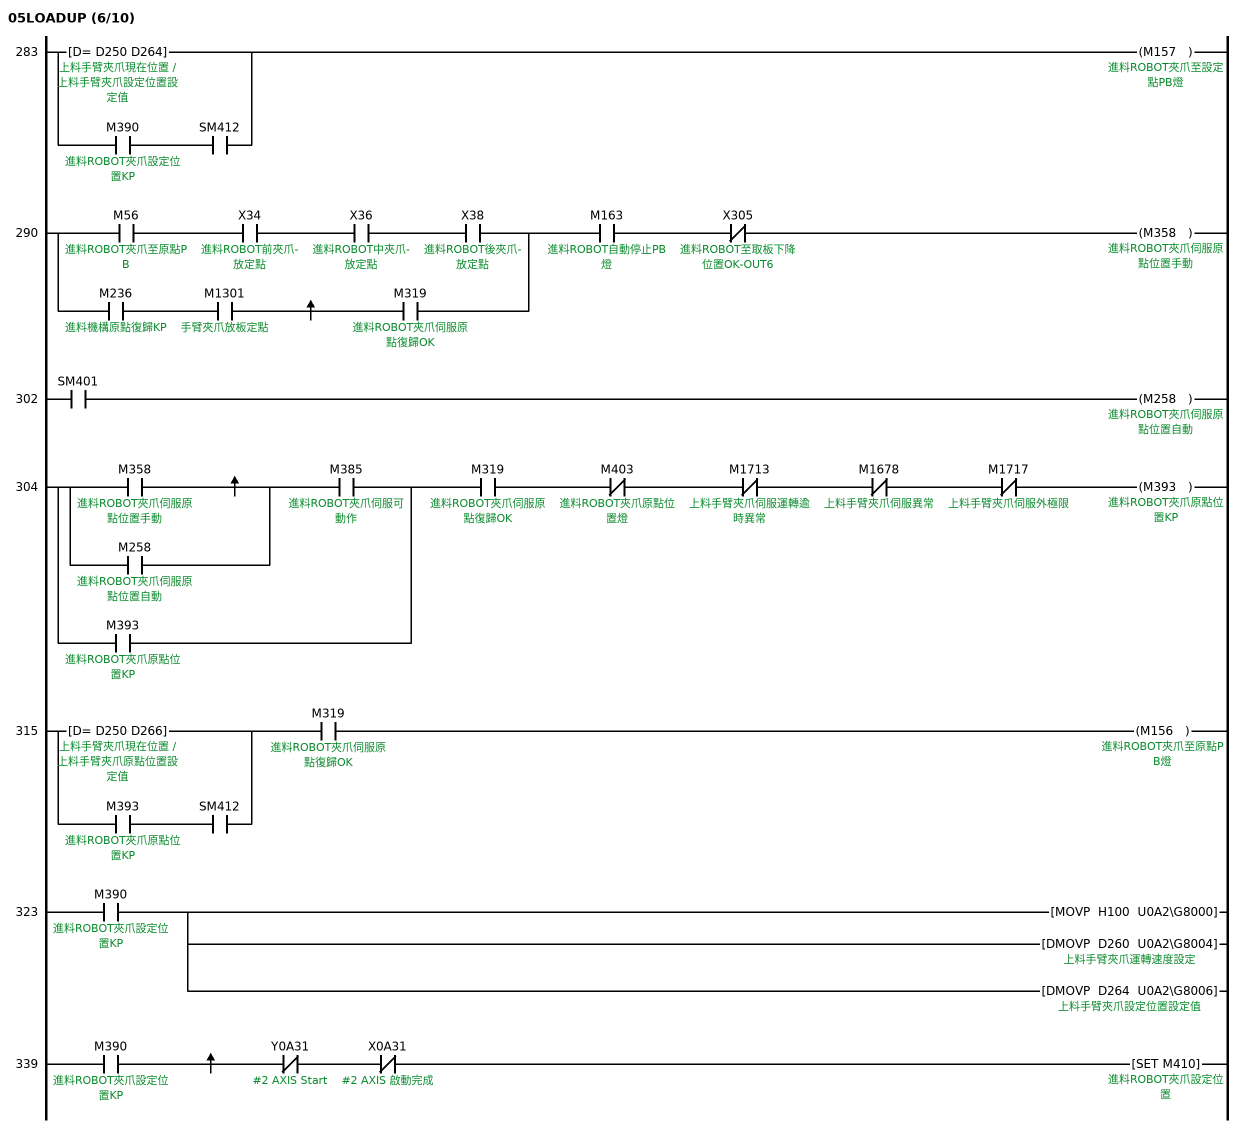
283   LDD=    D250 D264  ; 上料手臂夾爪現在位置 / 上料手臂夾爪設定位置設定值
      LD      M390  ; 進料ROBOT夾爪設定位置KP
      AND     SM412
      ORB
      OUT     M157  ; 進料ROBOT夾爪至設定點PB燈
290   LD      M56  ; 進料ROBOT夾爪至原點PB
      AND     X34  ; 進料ROBOT前夾爪-放定點
      AND     X36  ; 進料ROBOT中夾爪-放定點
      AND     X38  ; 進料ROBOT後夾爪-放定點
      LD      M236  ; 進料機構原點復歸KP
      AND     M1301  ; 手臂夾爪放板定點
      MEP
      AND     M319  ; 進料ROBOT夾爪伺服原點復歸OK
      ORB
      AND     M163  ; 進料ROBOT自動停止PB燈
      ANI     X305  ; 進料ROBOT至取板下降位置OK-OUT6
      OUT     M358  ; 進料ROBOT夾爪伺服原點位置手動
302   LD      SM401
      OUT     M258  ; 進料ROBOT夾爪伺服原點位置自動
304   LD      M358  ; 進料ROBOT夾爪伺服原點位置手動
      MEP
      OR      M258  ; 進料ROBOT夾爪伺服原點位置自動
      AND     M385  ; 進料ROBOT夾爪伺服可動作
      OR      M393  ; 進料ROBOT夾爪原點位置KP
      AND     M319  ; 進料ROBOT夾爪伺服原點復歸OK
      ANI     M403  ; 進料ROBOT夾爪原點位置燈
      ANI     M1713  ; 上料手臂夾爪伺服運轉逾時異常
      ANI     M1678  ; 上料手臂夾爪伺服異常
      ANI     M1717  ; 上料手臂夾爪伺服外極限
      OUT     M393  ; 進料ROBOT夾爪原點位置KP
315   LDD=    D250 D266  ; 上料手臂夾爪現在位置 / 上料手臂夾爪原點位置設定值
      LD      M393  ; 進料ROBOT夾爪原點位置KP
      AND     SM412
      ORB
      AND     M319  ; 進料ROBOT夾爪伺服原點復歸OK
      OUT     M156  ; 進料ROBOT夾爪至原點PB燈
323   LD      M390  ; 進料ROBOT夾爪設定位置KP
      MOVP    H100 U0A2\G8000
      DMOVP   D260 U0A2\G8004  ; 上料手臂夾爪運轉速度設定
      DMOVP   D264 U0A2\G8006
339   LD      M390  ; 進料ROBOT夾爪設定位置KP
      MEP
      ANI     Y0A31  ; #2 AXIS Start
      ANI     X0A31  ; #2 AXIS 啟動完成
      SET     M410  ; 進料ROBOT夾爪設定位置
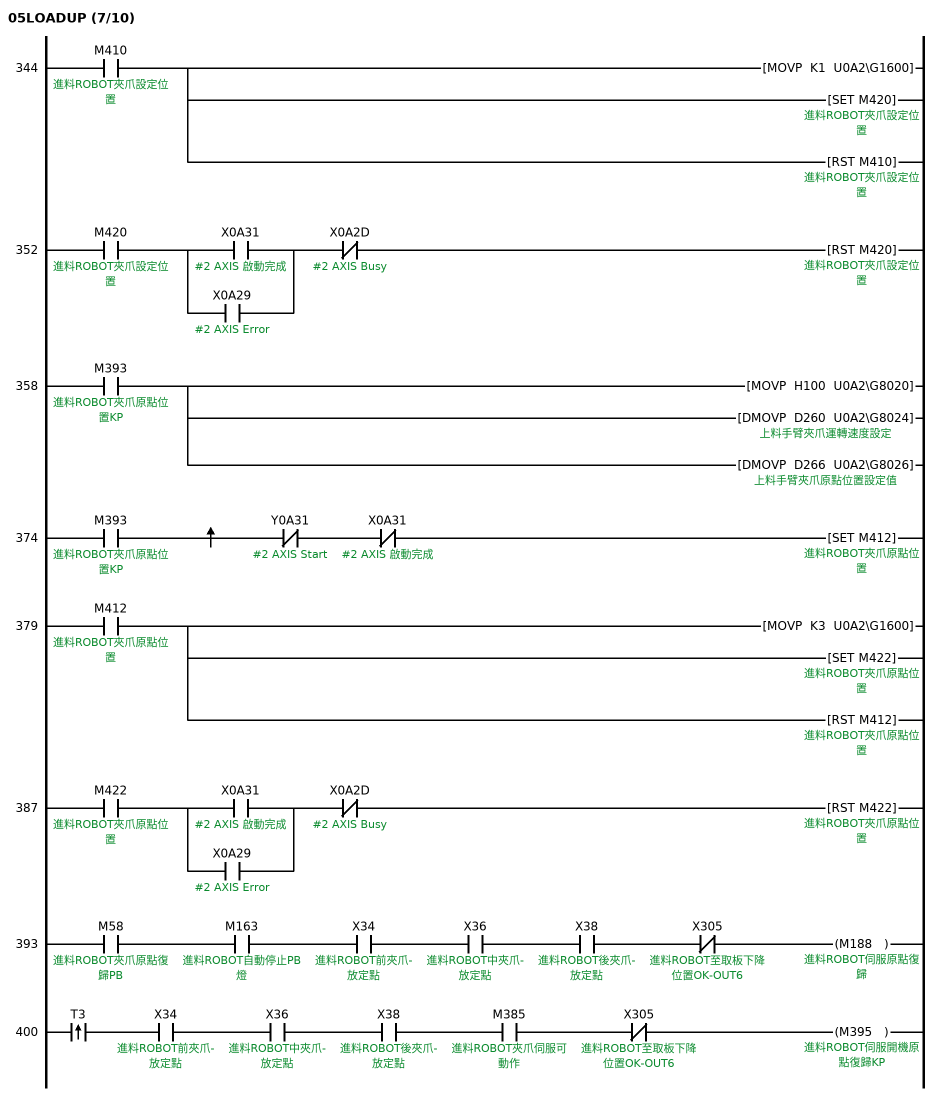
344   LD      M410  ; 進料ROBOT夾爪設定位置
      MOVP    K1 U0A2\G1600
      SET     M420  ; 進料ROBOT夾爪設定位置
      RST     M410  ; 進料ROBOT夾爪設定位置
352   LD      M420  ; 進料ROBOT夾爪設定位置
      LD      X0A31  ; #2 AXIS 啟動完成
      OR      X0A29  ; #2 AXIS Error
      ANB
      ANI     X0A2D  ; #2 AXIS Busy
      RST     M420  ; 進料ROBOT夾爪設定位置
358   LD      M393  ; 進料ROBOT夾爪原點位置KP
      MOVP    H100 U0A2\G8020
      DMOVP   D260 U0A2\G8024
      DMOVP   D266 U0A2\G8026
374   LD      M393  ; 進料ROBOT夾爪原點位置KP
      MEP
      ANI     Y0A31  ; #2 AXIS Start
      ANI     X0A31  ; #2 AXIS 啟動完成
      SET     M412  ; 進料ROBOT夾爪原點位置
379   LD      M412  ; 進料ROBOT夾爪原點位置
      MOVP    K3 U0A2\G1600
      SET     M422  ; 進料ROBOT夾爪原點位置
      RST     M412  ; 進料ROBOT夾爪原點位置
387   LD      M422  ; 進料ROBOT夾爪原點位置
      LD      X0A31  ; #2 AXIS 啟動完成
      OR      X0A29  ; #2 AXIS Error
      ANB
      ANI     X0A2D  ; #2 AXIS Busy
      RST     M422  ; 進料ROBOT夾爪原點位置
393   LD      M58  ; 進料ROBOT夾爪原點復歸PB
      AND     M163  ; 進料ROBOT自動停止PB燈
      AND     X34  ; 進料ROBOT前夾爪-放定點
      AND     X36  ; 進料ROBOT中夾爪-放定點
      AND     X38  ; 進料ROBOT後夾爪-放定點
      ANI     X305  ; 進料ROBOT至取板下降位置OK-OUT6
      OUT     M188  ; 進料ROBOT伺服原點復歸
400   LDP     T3
      AND     X34  ; 進料ROBOT前夾爪-放定點
      AND     X36  ; 進料ROBOT中夾爪-放定點
      AND     X38  ; 進料ROBOT後夾爪-放定點
      AND     M385  ; 進料ROBOT夾爪伺服可動作
      ANI     X305  ; 進料ROBOT至取板下降位置OK-OUT6
      OUT     M395  ; 進料ROBOT伺服開機原點復歸KP
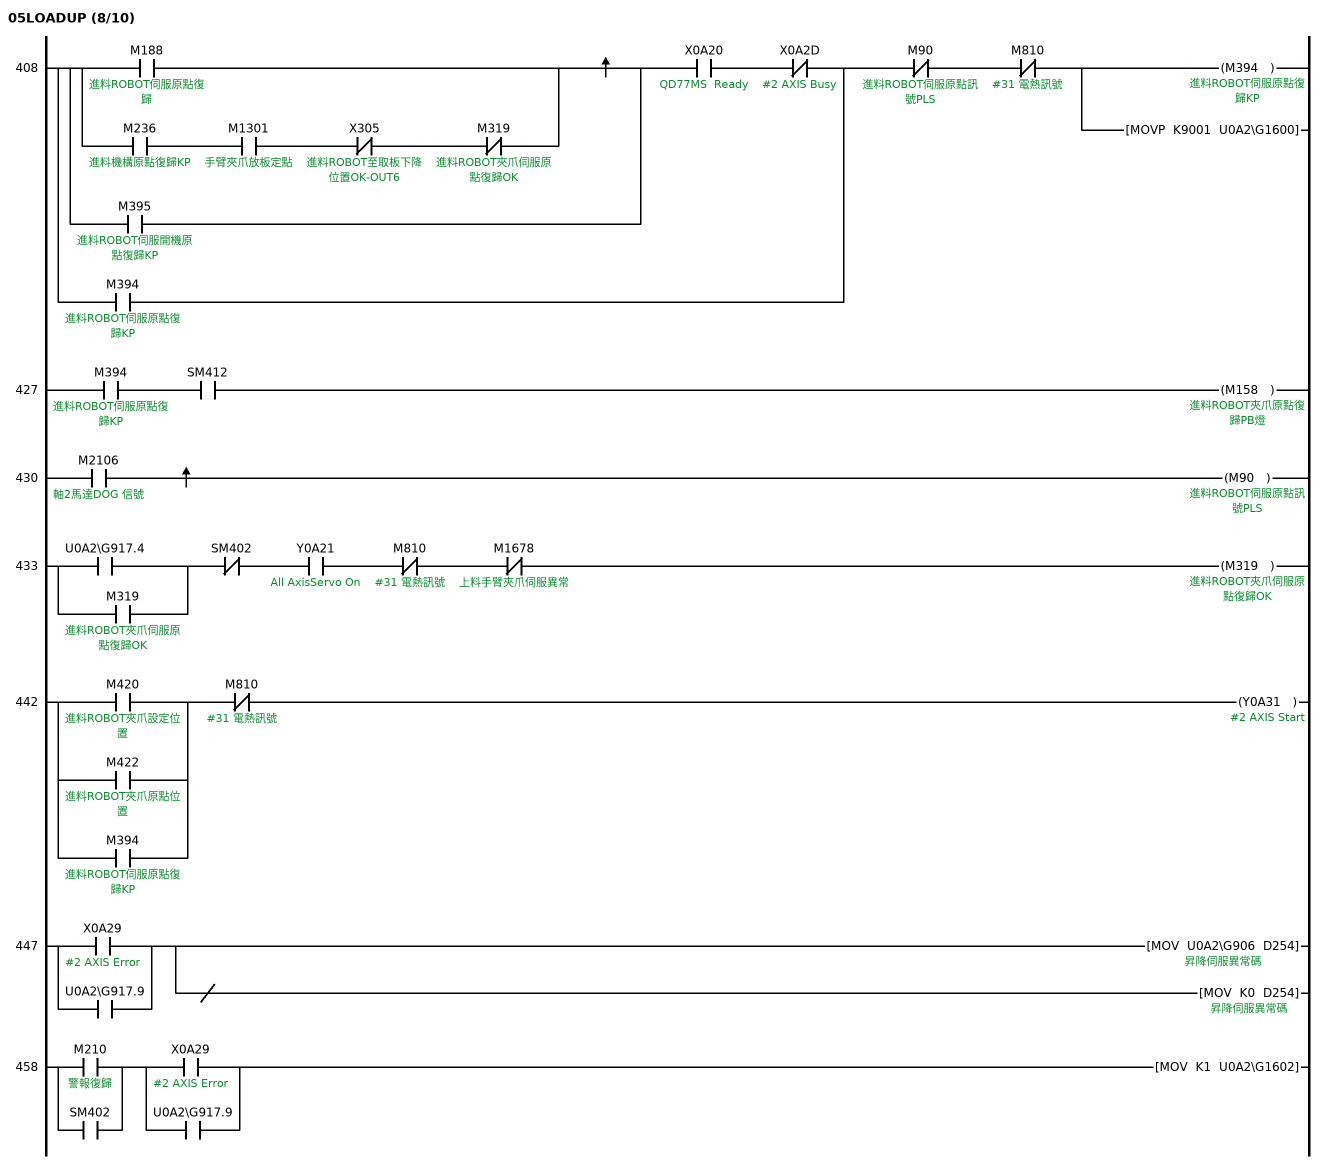
408   LD      M188  ; 進料ROBOT伺服原點復歸
      LD      M236  ; 進料機構原點復歸KP
      AND     M1301  ; 手臂夾爪放板定點
      ANI     X305  ; 進料ROBOT至取板下降位置OK-OUT6
      ANI     M319  ; 進料ROBOT夾爪伺服原點復歸OK
      ORB
      MEP
      OR      M395  ; 進料ROBOT伺服開機原點復歸KP
      AND     X0A20  ; QD77MS  Ready
      ANI     X0A2D  ; #2 AXIS Busy
      OR      M394  ; 進料ROBOT伺服原點復歸KP
      ANI     M90  ; 進料ROBOT伺服原點訊號PLS
      ANI     M810  ; #31 電熱訊號
      OUT     M394  ; 進料ROBOT伺服原點復歸KP
      MOVP    K9001 U0A2\G1600
427   LD      M394  ; 進料ROBOT伺服原點復歸KP
      AND     SM412
      OUT     M158  ; 進料ROBOT夾爪原點復歸PB燈
430   LD      M2106  ; 軸2馬達DOG 信號
      MEP
      OUT     M90  ; 進料ROBOT伺服原點訊號PLS
433   LD      U0A2\G917.4
      OR      M319  ; 進料ROBOT夾爪伺服原點復歸OK
      ANI     SM402
      AND     Y0A21  ; All AxisServo On
      ANI     M810  ; #31 電熱訊號
      ANI     M1678  ; 上料手臂夾爪伺服異常
      OUT     M319  ; 進料ROBOT夾爪伺服原點復歸OK
442   LD      M420  ; 進料ROBOT夾爪設定位置
      OR      M422  ; 進料ROBOT夾爪原點位置
      OR      M394  ; 進料ROBOT伺服原點復歸KP
      ANI     M810  ; #31 電熱訊號
      OUT     Y0A31  ; #2 AXIS Start
447   LD      X0A29  ; #2 AXIS Error
      OR      U0A2\G917.9
      MOV     U0A2\G906 D254  ; 昇降伺服異常碼
      INV
      MOV     K0 D254
458   LD      M210  ; 警報復歸
      OR      SM402
      LD      X0A29  ; #2 AXIS Error
      OR      U0A2\G917.9
      ANB
      MOV     K1 U0A2\G1602
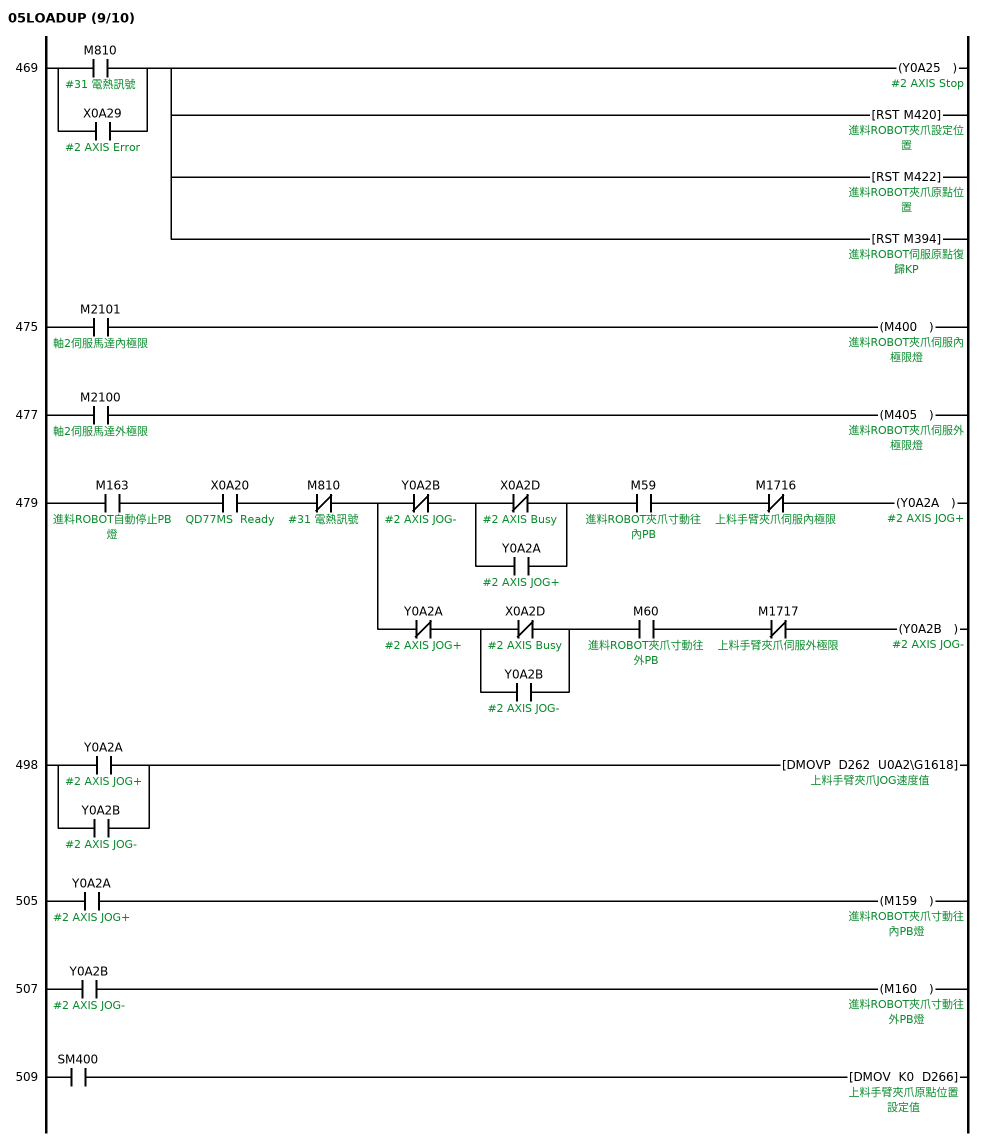
469   LD      M810  ; #31 電熱訊號
      OR      X0A29  ; #2 AXIS Error
      OUT     Y0A25  ; #2 AXIS Stop
      RST     M420  ; 進料ROBOT夾爪設定位置
      RST     M422  ; 進料ROBOT夾爪原點位置
      RST     M394  ; 進料ROBOT伺服原點復歸KP
475   LD      M2101  ; 軸2伺服馬達內極限
      OUT     M400  ; 進料ROBOT夾爪伺服內極限燈
477   LD      M2100  ; 軸2伺服馬達外極限
      OUT     M405  ; 進料ROBOT夾爪伺服外極限燈
479   LD      M163  ; 進料ROBOT自動停止PB燈
      AND     X0A20  ; QD77MS  Ready
      ANI     M810  ; #31 電熱訊號
      MPS
      ANI     Y0A2B  ; #2 AXIS JOG-
      LDI     X0A2D  ; #2 AXIS Busy
      OR      Y0A2A  ; #2 AXIS JOG+
      ANB
      AND     M59  ; 進料ROBOT夾爪寸動往內PB
      ANI     M1716  ; 上料手臂夾爪伺服內極限
      OUT     Y0A2A  ; #2 AXIS JOG+
      MPP
      ANI     Y0A2A  ; #2 AXIS JOG+
      LDI     X0A2D  ; #2 AXIS Busy
      OR      Y0A2B  ; #2 AXIS JOG-
      ANB
      AND     M60  ; 進料ROBOT夾爪寸動往外PB
      ANI     M1717  ; 上料手臂夾爪伺服外極限
      OUT     Y0A2B  ; #2 AXIS JOG-
498   LD      Y0A2A  ; #2 AXIS JOG+
      OR      Y0A2B  ; #2 AXIS JOG-
      DMOVP   D262 U0A2\G1618  ; 上料手臂夾爪JOG速度值
505   LD      Y0A2A  ; #2 AXIS JOG+
      OUT     M159  ; 進料ROBOT夾爪寸動往內PB燈
507   LD      Y0A2B  ; #2 AXIS JOG-
      OUT     M160  ; 進料ROBOT夾爪寸動往外PB燈
509   LD      SM400
      DMOV    K0 D266
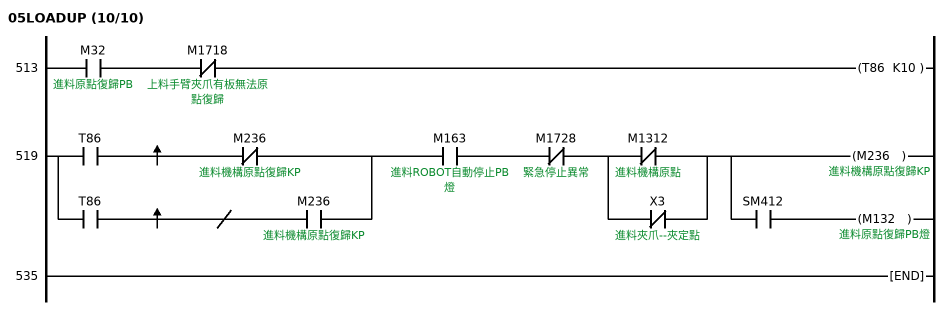
513   LD      M32  ; 進料原點復歸PB
      ANI     M1718  ; 上料手臂夾爪有板無法原點復歸
      OUT     T86 K10
519   LD      T86
      MEP
      ANI     M236  ; 進料機構原點復歸KP
      LD      T86
      MEP
      INV
      AND     M236  ; 進料機構原點復歸KP
      ORB
      AND     M163  ; 進料ROBOT自動停止PB燈
      ANI     M1728  ; 緊急停止異常
      LDI     M1312  ; 進料機構原點
      ORI     X3  ; 進料夾爪--夾定點
      ANB
      OUT     M236  ; 進料機構原點復歸KP
      AND     SM412
      OUT     M132  ; 進料原點復歸PB燈
535   END
END_PROGRAM

PROGRAM 06UNLOAD
